LIN {X 0,Y 361.896,Z 471.407,A -85,B 0,C 180,E1 -13251.652,E2 -13251.652} C_VEL
LIN {X 0,Y 361.932,Z 471.4,A -85,B 0,C 180,E1 -13255.29,E2 -13255.29} C_VEL
LIN {X 0,Y 361.912,Z 471.406,A -85,B 0,C 180,E1 -13257.779,E2 -13257.779} C_VEL
LIN {X 0,Y 361.841,Z 471.415,A -85,B 0,C 180,E1 -13261.629,E2 -13261.629} C_VEL
LIN {X 0,Y 361.878,Z 471.407,A -85,B 0,C 180,E1 -13265.344,E2 -13265.344} C_VEL
LIN {X 0,Y 361.873,Z 471.407,A -85,B 0,C 180,E1 -13269.026,E2 -13269.026} C_VEL
LIN {X 0,Y 361.839,Z 471.41,A -85,B 0,C 180,E1 -13272.828,E2 -13272.828} C_VEL
LIN {X 0,Y 361.819,Z 471.417,A -85,B 0,C 180,E1 -13275.6,E2 -13275.6} C_VEL
LIN {X 0,Y 361.188,Z 471.501,A -85,B 0,C 180,E1 -13276.53,E2 -13276.53} C_VEL
LIN {X 0,Y 358.309,Z 471.855,A -85,B 0,C 180,E1 -13278.041,E2 -13278.041} C_VEL
LIN {X 0,Y 355.876,Z 472.155,A -85,B 0,C 180,E1 -13279.265,E2 -13279.265} C_VEL
LIN {X 0,Y 354.876,Z 472.279,A -85,B 0,C 180,E1 -13280.212,E2 -13280.212} C_VEL
LIN {X 0,Y 354.821,Z 472.284,A -85,B 0,C 180,E1 -13280.532,E2 -13280.532} C_VEL
LIN {X 0,Y 354.824,Z 472.285,A -85,B 0,C 180,E1 -13284.3,E2 -13284.3} C_VEL
LIN {X 0,Y 354.789,Z 472.294,A -85,B 0,C 180,E1 -13287.666,E2 -13287.666} C_VEL
LIN {X 0,Y 354.87,Z 472.278,A -85,B 0,C 180,E1 -13290.621,E2 -13290.621} C_VEL
LIN {X 0,Y 354.901,Z 472.276,A -85,B 0,C 180,E1 -13294.172,E2 -13294.172} C_VEL
LIN {X 0,Y 354.836,Z 472.286,A -85,B 0,C 180,E1 -13297.894,E2 -13297.894} C_VEL
LIN {X 0,Y 354.924,Z 472.275,A -85,B 0,C 180,E1 -13301.891,E2 -13301.891} C_VEL
LIN {X 0,Y 354.944,Z 472.272,A -85,B 0,C 180,E1 -13305.981,E2 -13305.981} C_VEL
LIN {X 0,Y 354.979,Z 472.269,A -85,B 0,C 180,E1 -13309.736,E2 -13309.736} C_VEL
LIN {X 0,Y 355.115,Z 472.25,A -85,B 0,C 180,E1 -13312.037,E2 -13312.037} C_VEL
LIN {X 0,Y 355.093,Z 472.251,A -85,B 0,C 180,E1 -13314.32,E2 -13314.32} C_VEL
LIN {X 0,Y 355.246,Z 472.236,A -85,B 0,C 180,E1 -13317.732,E2 -13317.732} C_VEL
LIN {X 0,Y 355.398,Z 472.214,A -85,B 0,C 180,E1 -13320,E2 -13320} C_VEL
LIN {X 0,Y 355.244,Z 472.232,A -85,B 0,C 180,E1 -13322.267,E2 -13322.267} C_VEL
LIN {X 0,Y 355.139,Z 472.246,A -85,B 0,C 180,E1 -13326.819,E2 -13326.819} C_VEL
LIN {X 0,Y 355.015,Z 472.263,A -85,B 0,C 180,E1 -13329.112,E2 -13329.112} C_VEL
LIN {X 0,Y 354.921,Z 472.272,A -85,B 0,C 180,E1 -13332.581,E2 -13332.581} C_VEL
LIN {X 0,Y 354.89,Z 472.276,A -85,B 0,C 180,E1 -13336.096,E2 -13336.096} C_VEL
LIN {X 0,Y 354.901,Z 472.274,A -85,B 0,C 180,E1 -13338.472,E2 -13338.472} C_VEL
LIN {X 0,Y 354.835,Z 472.283,A -85,B 0,C 180,E1 -13342.106,E2 -13342.106} C_VEL
LIN {X 0,Y 354.899,Z 472.276,A -85,B 0,C 180,E1 -13345.827,E2 -13345.827} C_VEL
LIN {X 0,Y 354.817,Z 472.288,A -85,B 0,C 180,E1 -13349.682,E2 -13349.682} C_VEL
LIN {X 0,Y 354.805,Z 472.289,A -85,B 0,C 180,E1 -13353.702,E2 -13353.702} C_VEL
LIN {X 0,Y 354.801,Z 472.287,A -85,B 0,C 180,E1 -13356.459,E2 -13356.459} C_VEL
LIN {X 0,Y 354.824,Z 472.288,A -85,B 0,C 180,E1 -13359.424,E2 -13359.424} C_VEL
LIN {X 0,Y 354.835,Z 472.285,A -85,B 0,C 180,E1 -13362.876,E2 -13362.876} C_VEL
LIN {X 0,Y 354.861,Z 472.442,A -85,B 0,C 180,E1 -13365.478,E2 -13365.478} C_VEL
LIN {X 0,Y 356.023,Z 478.787,A -85,B 0,C 180,E1 -13369.351,E2 -13369.351} C_VEL
LIN {X 0,Y 357.063,Z 485.29,A -85,B 0,C 180,E1 -13373.108,E2 -13373.108} C_VEL
LIN {X 0,Y 356.927,Z 489.111,A -85,B 0,C 180,E1 -13375.179,E2 -13375.179} C_VEL
LIN {X 0,Y 356.106,Z 495.602,A -85,B 0,C 180,E1 -13378.579,E2 -13378.579} C_VEL
LIN {X 0,Y 355.345,Z 502.874,A -85,B 0,C 180,E1 -13382.305,E2 -13382.305} C_VEL
LIN {X 0,Y 354.675,Z 509.674,A -85,B 0,C 180,E1 -13385.714,E2 -13385.714} C_VEL
LIN {X 0,Y 354.097,Z 517.685,A -85,B 0,C 180,E1 -13389.676,E2 -13389.676} C_VEL
LIN {X 0,Y 353.998,Z 519.753,A -85,B 0,C 180,E1 -13390.691,E2 -13390.691} C_VEL
LIN {X 0,Y 355.817,Z 535.091,A -85,B 0,C 180,E1 -13391.457,E2 -13391.457} C_VEL
LIN {X 0,Y 357.371,Z 548.346,A -85,B 0,C 180,E1 -13392.345,E2 -13392.345} C_VEL
LIN {X 0,Y 357.95,Z 556.63,A -85,B 0,C 180,E1 -13393.019,E2 -13393.019} C_VEL
LIN {X 0,Y 357.02,Z 568.5,A -85,B 0,C 180,E1 -13394.15,E2 -13394.15} C_VEL
LIN {X 0,Y 356.03,Z 579.361,A -85,B 0,C 180,E1 -13395.443,E2 -13395.443} C_VEL
LIN {X 0,Y 355.222,Z 588.935,A -85,B 0,C 180,E1 -13396.849,E2 -13396.849} C_VEL
LIN {X 0,Y 354.587,Z 596.98,A -85,B 0,C 180,E1 -13398.279,E2 -13398.279} C_VEL
LIN {X 0,Y 354.005,Z 604.908,A -85,B 0,C 180,E1 -13399.997,E2 -13399.997} C_VEL
LIN {X 0,Y 353.691,Z 610.279,A -85,B 0,C 180,E1 -13401.43,E2 -13401.43} C_VEL
LIN {X 0,Y 353.5,Z 615.518,A -85,B 0,C 180,E1 -13403.149,E2 -13403.149} C_VEL
LIN {X 0,Y 353.454,Z 619.542,A -85,B 0,C 180,E1 -13404.867,E2 -13404.867} C_VEL
LIN {X 0,Y 353.343,Z 622.453,A -85,B 0,C 180,E1 -13406.579,E2 -13406.579} C_VEL
LIN {X 0,Y 353.477,Z 623.816,A -85,B 0,C 180,E1 -13407.721,E2 -13407.721} C_VEL
LIN {X 0,Y 353.476,Z 624.737,A -85,B 0,C 180,E1 -13408.861,E2 -13408.861} C_VEL
LIN {X 0,Y 353.463,Z 625.243,A -85,B 0,C 180,E1 -13410,E2 -13410} C_VEL
LIN {X 0,Y 353.464,Z 625.318,A -85,B 0,C 180,E1 -13411.14,E2 -13411.14} C_VEL
LIN {X 0,Y 353.371,Z 624.931,A -85,B 0,C 180,E1 -13412.28,E2 -13412.28} C_VEL
LIN {X 0,Y 353.322,Z 622.937,A -85,B 0,C 180,E1 -13414.564,E2 -13414.564} C_VEL
LIN {X 0,Y 353.314,Z 620.847,A -85,B 0,C 180,E1 -13415.966,E2 -13415.966} C_VEL
LIN {X 0,Y 353.604,Z 616.652,A -85,B 0,C 180,E1 -13417.998,E2 -13417.998} C_VEL
LIN {X 0,Y 353.981,Z 611.938,A -85,B 0,C 180,E1 -13419.716,E2 -13419.716} C_VEL
LIN {X 0,Y 354.771,Z 604.943,A -85,B 0,C 180,E1 -13421.716,E2 -13421.716} C_VEL
LIN {X 0,Y 355.788,Z 597.461,A -85,B 0,C 180,E1 -13423.421,E2 -13423.421} C_VEL
LIN {X 0,Y 356.862,Z 588.946,A -85,B 0,C 180,E1 -13425.028,E2 -13425.028} C_VEL
LIN {X 0,Y 358.555,Z 578.253,A -85,B 0,C 180,E1 -13426.659,E2 -13426.659} C_VEL
LIN {X 0,Y 360.253,Z 567.141,A -85,B 0,C 180,E1 -13428.041,E2 -13428.041} C_VEL
LIN {X 0,Y 361.219,Z 559.295,A -85,B 0,C 180,E1 -13428.873,E2 -13428.873} C_VEL
LIN {X 0,Y 361.174,Z 546.774,A -85,B 0,C 180,E1 -13430.1,E2 -13430.1} C_VEL
LIN {X 0,Y 359.932,Z 535.75,A -85,B 0,C 180,E1 -13431.118,E2 -13431.118} C_VEL
LIN {X 0,Y 357.617,Z 524.701,A -85,B 0,C 180,E1 -13432.098,E2 -13432.098} C_VEL
LIN {X 0,Y 355.357,Z 517.035,A -85,B 0,C 180,E1 -13432.792,E2 -13432.792} C_VEL
LIN {X 0,Y 354.616,Z 513.908,A -85,B 0,C 180,E1 -13433.055,E2 -13433.055} C_VEL
LIN {X 0,Y 355.282,Z 507.666,A -85,B 0,C 180,E1 -13436.429,E2 -13436.429} C_VEL
LIN {X 0,Y 356.057,Z 502.051,A -85,B 0,C 180,E1 -13439.716,E2 -13439.716} C_VEL
LIN {X 0,Y 356.726,Z 498.243,A -85,B 0,C 180,E1 -13442.137,E2 -13442.137} C_VEL
LIN {X 0,Y 357.445,Z 494.507,A -85,B 0,C 180,E1 -13444.764,E2 -13444.764} C_VEL
LIN {X 0,Y 357.796,Z 492.467,A -85,B 0,C 180,E1 -13446.357,E2 -13446.357} C_VEL
LIN {X 0,Y 357.78,Z 489.641,A -85,B 0,C 180,E1 -13448.946,E2 -13448.946} C_VEL
LIN {X 0,Y 357.413,Z 487.044,A -85,B 0,C 180,E1 -13451.956,E2 -13451.956} C_VEL
LIN {X 0,Y 357.086,Z 485.013,A -85,B 0,C 180,E1 -13455.116,E2 -13455.116} C_VEL
LIN {X 0,Y 356.777,Z 483.627,A -85,B 0,C 180,E1 -13458.465,E2 -13458.465} C_VEL
LIN {X 0,Y 356.561,Z 482.938,A -85,B 0,C 180,E1 -13462.039,E2 -13462.039} C_VEL
LIN {X 0,Y 356.269,Z 482.954,A -85,B 0,C 180,E1 -13465.105,E2 -13465.105} C_VEL
LIN {X 0,Y 355.925,Z 483.444,A -85,B 0,C 180,E1 -13468.111,E2 -13468.111} C_VEL
LIN {X 0,Y 355.416,Z 484.534,A -85,B 0,C 180,E1 -13471.668,E2 -13471.668} C_VEL
LIN {X 0,Y 354.986,Z 486.226,A -85,B 0,C 180,E1 -13475.604,E2 -13475.604} C_VEL
LIN {X 0,Y 354.856,Z 487.017,A -85,B 0,C 180,E1 -13477.145,E2 -13477.145} C_VEL
LIN {X 0,Y 355.852,Z 489.82,A -85,B 0,C 180,E1 -13477.439,E2 -13477.439} C_VEL
LIN {X 0,Y 357.99,Z 494.025,A -85,B 0,C 180,E1 -13477.965,E2 -13477.965} C_VEL
LIN {X 0,Y 361.932,Z 504.222,A -85,B 0,C 180,E1 -13479.157,E2 -13479.157} C_VEL
LIN {X 0,Y 364.472,Z 513.793,A -85,B 0,C 180,E1 -13480.259,E2 -13480.259} C_VEL
LIN {X 0,Y 364.253,Z 518.028,A -85,B 0,C 180,E1 -13480.651,E2 -13480.651} C_VEL
LIN {X 0,Y 362.785,Z 529.035,A -85,B 0,C 180,E1 -13481.74,E2 -13481.74} C_VEL
LIN {X 0,Y 361.233,Z 539.619,A -85,B 0,C 180,E1 -13483.032,E2 -13483.032} C_VEL
LIN {X 0,Y 359.697,Z 548.878,A -85,B 0,C 180,E1 -13484.416,E2 -13484.416} C_VEL
LIN {X 0,Y 358.425,Z 556.592,A -85,B 0,C 180,E1 -13485.812,E2 -13485.812} C_VEL
LIN {X 0,Y 357.08,Z 564.286,A -85,B 0,C 180,E1 -13487.497,E2 -13487.497} C_VEL
LIN {X 0,Y 356.143,Z 570.486,A -85,B 0,C 180,E1 -13489.195,E2 -13489.195} C_VEL
LIN {X 0,Y 355.273,Z 575.452,A -85,B 0,C 180,E1 -13490.895,E2 -13490.895} C_VEL
LIN {X 0,Y 354.489,Z 579.713,A -85,B 0,C 180,E1 -13492.792,E2 -13492.792} C_VEL
LIN {X 0,Y 354.101,Z 582.167,A -85,B 0,C 180,E1 -13494.305,E2 -13494.305} C_VEL
LIN {X 0,Y 354.036,Z 583.522,A -85,B 0,C 180,E1 -13495.446,E2 -13495.446} C_VEL
LIN {X 0,Y 353.821,Z 584.446,A -85,B 0,C 180,E1 -13496.584,E2 -13496.584} C_VEL
LIN {X 0,Y 353.65,Z 584.978,A -85,B 0,C 180,E1 -13497.722,E2 -13497.722} C_VEL
LIN {X 0,Y 353.526,Z 585.118,A -85,B 0,C 180,E1 -13498.861,E2 -13498.861} C_VEL
LIN {X 0,Y 353.466,Z 584.834,A -85,B 0,C 180,E1 -13500,E2 -13500} C_VEL
LIN {X 0,Y 353.486,Z 584.117,A -85,B 0,C 180,E1 -13501.14,E2 -13501.14} C_VEL
LIN {X 0,Y 353.519,Z 583.003,A -85,B 0,C 180,E1 -13502.279,E2 -13502.279} C_VEL
LIN {X 0,Y 353.539,Z 580.526,A -85,B 0,C 180,E1 -13503.99,E2 -13503.99} C_VEL
LIN {X 0,Y 353.757,Z 577.033,A -85,B 0,C 180,E1 -13505.701,E2 -13505.701} C_VEL
LIN {X 0,Y 354.05,Z 572.439,A -85,B 0,C 180,E1 -13507.413,E2 -13507.413} C_VEL
LIN {X 0,Y 354.437,Z 566.619,A -85,B 0,C 180,E1 -13509.128,E2 -13509.128} C_VEL
LIN {X 0,Y 355.01,Z 559.372,A -85,B 0,C 180,E1 -13510.84,E2 -13510.84} C_VEL
LIN {X 0,Y 355.731,Z 550.381,A -85,B 0,C 180,E1 -13512.552,E2 -13512.552} C_VEL
LIN {X 0,Y 356.656,Z 540.246,A -85,B 0,C 180,E1 -13514.114,E2 -13514.114} C_VEL
LIN {X 0,Y 357.475,Z 529.945,A -85,B 0,C 180,E1 -13515.402,E2 -13515.402} C_VEL
LIN {X 0,Y 358.342,Z 517.407,A -85,B 0,C 180,E1 -13516.669,E2 -13516.669} C_VEL
LIN {X 0,Y 359.063,Z 507.592,A -85,B 0,C 180,E1 -13517.458,E2 -13517.458} C_VEL
LIN {X 0,Y 357.067,Z 496.682,A -85,B 0,C 180,E1 -13518.254,E2 -13518.254} C_VEL
LIN {X 0,Y 354.036,Z 482.545,A -85,B 0,C 180,E1 -13519.063,E2 -13519.063} C_VEL
LIN {X 0,Y 353.631,Z 480.363,A -85,B 0,C 180,E1 -13519.199,E2 -13519.199} C_VEL
LIN {X 0,Y 353.639,Z 477.42,A -85,B 0,C 180,E1 -13522.185,E2 -13522.185} C_VEL
LIN {X 0,Y 353.81,Z 473.84,A -85,B 0,C 180,E1 -13525.913,E2 -13525.913} C_VEL
LIN {X 0,Y 353.84,Z 472.639,A -85,B 0,C 180,E1 -13527.183,E2 -13527.183} C_VEL
LIN {X 0,Y 354.095,Z 472.378,A -85,B 0,C 180,E1 -13529.749,E2 -13529.749} C_VEL
LIN {X 0,Y 354.394,Z 472.343,A -85,B 0,C 180,E1 -13532.374,E2 -13532.374} C_VEL
LIN {X 0,Y 354.715,Z 472.299,A -85,B 0,C 180,E1 -13535.675,E2 -13535.675} C_VEL
LIN {X 0,Y 354.797,Z 472.29,A -85,B 0,C 180,E1 -13537.885,E2 -13537.885} C_VEL
LIN {X 0,Y 354.792,Z 472.288,A -85,B 0,C 180,E1 -13541.172,E2 -13541.172} C_VEL
LIN {X 0,Y 354.768,Z 472.294,A -85,B 0,C 180,E1 -13544.507,E2 -13544.507} C_VEL
LIN {X 0,Y 354.799,Z 472.288,A -85,B 0,C 180,E1 -13547.663,E2 -13547.663} C_VEL
LIN {X 0,Y 354.819,Z 472.287,A -85,B 0,C 180,E1 -13550.666,E2 -13550.666} C_VEL
LIN {X 0,Y 354.827,Z 472.288,A -85,B 0,C 180,E1 -13554.301,E2 -13554.301} C_VEL
LIN {X 0,Y 354.792,Z 472.29,A -85,B 0,C 180,E1 -13557.667,E2 -13557.667} C_VEL
LIN {X 0,Y 354.851,Z 472.282,A -85,B 0,C 180,E1 -13561.619,E2 -13561.619} C_VEL
LIN {X 0,Y 354.904,Z 472.279,A -85,B 0,C 180,E1 -13564.173,E2 -13564.173} C_VEL
LIN {X 0,Y 354.84,Z 472.285,A -85,B 0,C 180,E1 -13567.894,E2 -13567.894} C_VEL
LIN {X 0,Y 354.928,Z 472.275,A -85,B 0,C 180,E1 -13571.891,E2 -13571.891} C_VEL
LIN {X 0,Y 354.948,Z 472.274,A -85,B 0,C 180,E1 -13575.981,E2 -13575.981} C_VEL
LIN {X 0,Y 354.982,Z 472.268,A -85,B 0,C 180,E1 -13579.736,E2 -13579.736} C_VEL
LIN {X 0,Y 355.125,Z 472.246,A -85,B 0,C 180,E1 -13583.18,E2 -13583.18} C_VEL
LIN {X 0,Y 355.249,Z 472.235,A -85,B 0,C 180,E1 -13587.732,E2 -13587.732} C_VEL
LIN {X 0,Y 355.401,Z 472.217,A -85,B 0,C 180,E1 -13590,E2 -13590} C_VEL
LIN {X 0,Y 355.249,Z 472.235,A -85,B 0,C 180,E1 -13592.267,E2 -13592.267} C_VEL
LIN {X 0,Y 355.108,Z 472.248,A -85,B 0,C 180,E1 -13596.82,E2 -13596.82} C_VEL
LIN {X 0,Y 354.983,Z 472.267,A -85,B 0,C 180,E1 -13600.264,E2 -13600.264} C_VEL
LIN {X 0,Y 354.947,Z 472.273,A -85,B 0,C 180,E1 -13604.019,E2 -13604.019} C_VEL
LIN {X 0,Y 354.927,Z 472.275,A -85,B 0,C 180,E1 -13608.108,E2 -13608.108} C_VEL
LIN {X 0,Y 354.839,Z 472.286,A -85,B 0,C 180,E1 -13612.106,E2 -13612.106} C_VEL
LIN {X 0,Y 354.903,Z 472.279,A -85,B 0,C 180,E1 -13615.827,E2 -13615.827} C_VEL
LIN {X 0,Y 354.821,Z 472.289,A -85,B 0,C 180,E1 -13619.681,E2 -13619.681} C_VEL
LIN {X 0,Y 354.809,Z 472.29,A -85,B 0,C 180,E1 -13623.702,E2 -13623.702} C_VEL
LIN {X 0,Y 354.804,Z 472.287,A -85,B 0,C 180,E1 -13626.458,E2 -13626.458} C_VEL
LIN {X 0,Y 354.826,Z 472.287,A -85,B 0,C 180,E1 -13629.423,E2 -13629.423} C_VEL
LIN {X 0,Y 354.791,Z 472.288,A -85,B 0,C 180,E1 -13632.867,E2 -13632.867} C_VEL
LIN {X 0,Y 354.771,Z 472.294,A -85,B 0,C 180,E1 -13636.103,E2 -13636.103} C_VEL
LIN {X 0,Y 354.79,Z 472.289,A -85,B 0,C 180,E1 -13639.179,E2 -13639.179} C_VEL
LIN {X 0,Y 354.821,Z 472.284,A -85,B 0,C 180,E1 -13640.532,E2 -13640.532} C_VEL
LIN {X 0,Y 354.218,Z 472.366,A -85,B 0,C 180,E1 -13641.48,E2 -13641.48} C_VEL
LIN {X 0,Y 351.361,Z 472.727,A -85,B 0,C 180,E1 -13643.02,E2 -13643.02} C_VEL
LIN {X 0,Y 348.896,Z 473.032,A -85,B 0,C 180,E1 -13644.267,E2 -13644.267} C_VEL
LIN {X 0,Y 347.832,Z 473.161,A -85,B 0,C 180,E1 -13645.232,E2 -13645.232} C_VEL
LIN {X 0,Y 347.746,Z 473.17,A -85,B 0,C 180,E1 -13645.559,E2 -13645.559} C_VEL
LIN {X 0,Y 347.765,Z 473.168,A -85,B 0,C 180,E1 -13649.653,E2 -13649.653} C_VEL
LIN {X 0,Y 347.853,Z 473.152,A -85,B 0,C 180,E1 -13652.744,E2 -13652.744} C_VEL
LIN {X 0,Y 347.79,Z 473.162,A -85,B 0,C 180,E1 -13656.162,E2 -13656.162} C_VEL
LIN {X 0,Y 347.819,Z 473.159,A -85,B 0,C 180,E1 -13659.909,E2 -13659.909} C_VEL
LIN {X 0,Y 347.868,Z 473.151,A -85,B 0,C 180,E1 -13662.359,E2 -13662.359} C_VEL
LIN {X 0,Y 347.898,Z 473.149,A -85,B 0,C 180,E1 -13665.97,E2 -13665.97} C_VEL
LIN {X 0,Y 347.929,Z 473.148,A -85,B 0,C 180,E1 -13669.525,E2 -13669.525} C_VEL
LIN {X 0,Y 348.075,Z 473.128,A -85,B 0,C 180,E1 -13671.874,E2 -13671.874} C_VEL
LIN {X 0,Y 348.068,Z 473.126,A -85,B 0,C 180,E1 -13674.205,E2 -13674.205} C_VEL
LIN {X 0,Y 348.209,Z 473.112,A -85,B 0,C 180,E1 -13677.686,E2 -13677.686} C_VEL
LIN {X 0,Y 348.347,Z 473.092,A -85,B 0,C 180,E1 -13680,E2 -13680} C_VEL
LIN {X 0,Y 348.207,Z 473.108,A -85,B 0,C 180,E1 -13682.313,E2 -13682.313} C_VEL
LIN {X 0,Y 348.107,Z 473.122,A -85,B 0,C 180,E1 -13686.957,E2 -13686.957} C_VEL
LIN {X 0,Y 347.968,Z 473.142,A -85,B 0,C 180,E1 -13689.298,E2 -13689.298} C_VEL
LIN {X 0,Y 347.89,Z 473.149,A -85,B 0,C 180,E1 -13692.839,E2 -13692.839} C_VEL
LIN {X 0,Y 347.839,Z 473.154,A -85,B 0,C 180,E1 -13696.431,E2 -13696.431} C_VEL
LIN {X 0,Y 347.851,Z 473.154,A -85,B 0,C 180,E1 -13698.86,E2 -13698.86} C_VEL
LIN {X 0,Y 347.774,Z 473.162,A -85,B 0,C 180,E1 -13702.579,E2 -13702.579} C_VEL
LIN {X 0,Y 347.813,Z 473.16,A -85,B 0,C 180,E1 -13705.108,E2 -13705.108} C_VEL
LIN {X 0,Y 347.808,Z 473.161,A -85,B 0,C 180,E1 -13707.694,E2 -13707.694} C_VEL
LIN {X 0,Y 347.749,Z 473.165,A -85,B 0,C 180,E1 -13710.348,E2 -13710.348} C_VEL
LIN {X 0,Y 347.748,Z 473.166,A -85,B 0,C 180,E1 -13714.044,E2 -13714.044} C_VEL
LIN {X 0,Y 347.766,Z 473.168,A -85,B 0,C 180,E1 -13717.32,E2 -13717.32} C_VEL
LIN {X 0,Y 347.793,Z 473.16,A -85,B 0,C 180,E1 -13720.289,E2 -13720.289} C_VEL
LIN {X 0,Y 347.786,Z 473.166,A -85,B 0,C 180,E1 -13723.398,E2 -13723.398} C_VEL
LIN {X 0,Y 347.86,Z 473.23,A -85,B 0,C 180,E1 -13725.206,E2 -13725.206} C_VEL
LIN {X 0,Y 348.936,Z 479.491,A -85,B 0,C 180,E1 -13729.112,E2 -13729.112} C_VEL
LIN {X 0,Y 349.857,Z 484.863,A -85,B 0,C 180,E1 -13732.299,E2 -13732.299} C_VEL
LIN {X 0,Y 349.979,Z 488.554,A -85,B 0,C 180,E1 -13734.384,E2 -13734.384} C_VEL
LIN {X 0,Y 349.225,Z 494.695,A -85,B 0,C 180,E1 -13737.697,E2 -13737.697} C_VEL
LIN {X 0,Y 348.389,Z 502.297,A -85,B 0,C 180,E1 -13741.702,E2 -13741.702} C_VEL
LIN {X 0,Y 347.642,Z 509.619,A -85,B 0,C 180,E1 -13745.468,E2 -13745.468} C_VEL
LIN {X 0,Y 346.993,Z 518.291,A -85,B 0,C 180,E1 -13749.86,E2 -13749.86} C_VEL
LIN {X 0,Y 346.912,Z 519.429,A -85,B 0,C 180,E1 -13750.434,E2 -13750.434} C_VEL
LIN {X 0,Y 348.644,Z 534.247,A -85,B 0,C 180,E1 -13751.184,E2 -13751.184} C_VEL
LIN {X 0,Y 350.184,Z 547.739,A -85,B 0,C 180,E1 -13752.107,E2 -13752.107} C_VEL
LIN {X 0,Y 350.889,Z 557.922,A -85,B 0,C 180,E1 -13752.967,E2 -13752.967} C_VEL
LIN {X 0,Y 349.929,Z 569.441,A -85,B 0,C 180,E1 -13754.119,E2 -13754.119} C_VEL
LIN {X 0,Y 348.815,Z 580.976,A -85,B 0,C 180,E1 -13755.572,E2 -13755.572} C_VEL
LIN {X 0,Y 348.09,Z 589.406,A -85,B 0,C 180,E1 -13756.872,E2 -13756.872} C_VEL
LIN {X 0,Y 347.451,Z 597.304,A -85,B 0,C 180,E1 -13758.33,E2 -13758.33} C_VEL
LIN {X 0,Y 346.91,Z 605.057,A -85,B 0,C 180,E1 -13760.084,E2 -13760.084} C_VEL
LIN {X 0,Y 346.541,Z 611.261,A -85,B 0,C 180,E1 -13761.839,E2 -13761.839} C_VEL
LIN {X 0,Y 346.342,Z 616.887,A -85,B 0,C 180,E1 -13763.887,E2 -13763.887} C_VEL
LIN {X 0,Y 346.366,Z 619.905,A -85,B 0,C 180,E1 -13765.345,E2 -13765.345} C_VEL
LIN {X 0,Y 346.266,Z 621.792,A -85,B 0,C 180,E1 -13766.509,E2 -13766.509} C_VEL
LIN {X 0,Y 346.397,Z 623.234,A -85,B 0,C 180,E1 -13767.675,E2 -13767.675} C_VEL
LIN {X 0,Y 346.414,Z 624.197,A -85,B 0,C 180,E1 -13768.838,E2 -13768.838} C_VEL
LIN {X 0,Y 346.399,Z 624.74,A -85,B 0,C 180,E1 -13770,E2 -13770} C_VEL
LIN {X 0,Y 346.4,Z 624.872,A -85,B 0,C 180,E1 -13771.163,E2 -13771.163} C_VEL
LIN {X 0,Y 346.272,Z 624.543,A -85,B 0,C 180,E1 -13772.327,E2 -13772.327} C_VEL
LIN {X 0,Y 346.215,Z 623.786,A -85,B 0,C 180,E1 -13773.492,E2 -13773.492} C_VEL
LIN {X 0,Y 346.233,Z 622.625,A -85,B 0,C 180,E1 -13774.657,E2 -13774.657} C_VEL
LIN {X 0,Y 346.242,Z 620.845,A -85,B 0,C 180,E1 -13775.957,E2 -13775.957} C_VEL
LIN {X 0,Y 346.544,Z 616.518,A -85,B 0,C 180,E1 -13778.162,E2 -13778.162} C_VEL
LIN {X 0,Y 346.965,Z 611.913,A -85,B 0,C 180,E1 -13779.914,E2 -13779.914} C_VEL
LIN {X 0,Y 347.817,Z 605.087,A -85,B 0,C 180,E1 -13781.953,E2 -13781.953} C_VEL
LIN {X 0,Y 348.887,Z 597.774,A -85,B 0,C 180,E1 -13783.692,E2 -13783.692} C_VEL
LIN {X 0,Y 350.175,Z 588.755,A -85,B 0,C 180,E1 -13785.451,E2 -13785.451} C_VEL
LIN {X 0,Y 351.97,Z 578.118,A -85,B 0,C 180,E1 -13787.129,E2 -13787.129} C_VEL
LIN {X 0,Y 353.797,Z 567.069,A -85,B 0,C 180,E1 -13788.532,E2 -13788.532} C_VEL
LIN {X 0,Y 354.704,Z 559.366,A -85,B 0,C 180,E1 -13789.383,E2 -13789.383} C_VEL
LIN {X 0,Y 354.764,Z 547.801,A -85,B 0,C 180,E1 -13790.583,E2 -13790.583} C_VEL
LIN {X 0,Y 353.472,Z 536.234,A -85,B 0,C 180,E1 -13791.711,E2 -13791.711} C_VEL
LIN {X 0,Y 350.89,Z 524.202,A -85,B 0,C 180,E1 -13792.878,E2 -13792.878} C_VEL
LIN {X 0,Y 348.41,Z 516.176,A -85,B 0,C 180,E1 -13793.663,E2 -13793.663} C_VEL
LIN {X 0,Y 347.741,Z 513.187,A -85,B 0,C 180,E1 -13793.94,E2 -13793.94} C_VEL
LIN {X 0,Y 348.508,Z 506.68,A -85,B 0,C 180,E1 -13797.634,E2 -13797.634} C_VEL
LIN {X 0,Y 349.533,Z 500.482,A -85,B 0,C 180,E1 -13801.519,E2 -13801.519} C_VEL
LIN {X 0,Y 350.446,Z 496.008,A -85,B 0,C 180,E1 -13804.691,E2 -13804.691} C_VEL
LIN {X 0,Y 350.87,Z 493.249,A -85,B 0,C 180,E1 -13806.935,E2 -13806.935} C_VEL
LIN {X 0,Y 350.879,Z 491.449,A -85,B 0,C 180,E1 -13808.633,E2 -13808.633} C_VEL
LIN {X 0,Y 350.474,Z 488.488,A -85,B 0,C 180,E1 -13812.102,E2 -13812.102} C_VEL
LIN {X 0,Y 350.142,Z 486.451,A -85,B 0,C 180,E1 -13815.371,E2 -13815.371} C_VEL
LIN {X 0,Y 349.864,Z 485.181,A -85,B 0,C 180,E1 -13818.479,E2 -13818.479} C_VEL
LIN {X 0,Y 349.634,Z 484.512,A -85,B 0,C 180,E1 -13821.623,E2 -13821.623} C_VEL
LIN {X 0,Y 349.398,Z 484.393,A -85,B 0,C 180,E1 -13824.315,E2 -13824.315} C_VEL
LIN {X 0,Y 349.006,Z 484.796,A -85,B 0,C 180,E1 -13827.754,E2 -13827.754} C_VEL
LIN {X 0,Y 348.523,Z 485.683,A -85,B 0,C 180,E1 -13831.056,E2 -13831.056} C_VEL
LIN {X 0,Y 348.058,Z 487.19,A -85,B 0,C 180,E1 -13834.911,E2 -13834.911} C_VEL
LIN {X 0,Y 347.955,Z 487.974,A -85,B 0,C 180,E1 -13836.278,E2 -13836.278} C_VEL
LIN {X 0,Y 349.083,Z 490.882,A -85,B 0,C 180,E1 -13836.62,E2 -13836.62} C_VEL
LIN {X 0,Y 350.066,Z 492.672,A -85,B 0,C 180,E1 -13836.876,E2 -13836.876} C_VEL
LIN {X 0,Y 354.719,Z 503.244,A -85,B 0,C 180,E1 -13838.251,E2 -13838.251} C_VEL
LIN {X 0,Y 357.709,Z 513.477,A -85,B 0,C 180,E1 -13839.507,E2 -13839.507} C_VEL
LIN {X 0,Y 358.384,Z 516.83,A -85,B 0,C 180,E1 -13839.915,E2 -13839.915} C_VEL
LIN {X 0,Y 356.794,Z 528.176,A -85,B 0,C 180,E1 -13841.033,E2 -13841.033} C_VEL
LIN {X 0,Y 355.113,Z 538.661,A -85,B 0,C 180,E1 -13842.316,E2 -13842.316} C_VEL
LIN {X 0,Y 353.335,Z 548.893,A -85,B 0,C 180,E1 -13843.831,E2 -13843.831} C_VEL
LIN {X 0,Y 351.892,Z 556.682,A -85,B 0,C 180,E1 -13845.248,E2 -13845.248} C_VEL
LIN {X 0,Y 350.485,Z 564.358,A -85,B 0,C 180,E1 -13846.963,E2 -13846.963} C_VEL
LIN {X 0,Y 349.262,Z 571.565,A -85,B 0,C 180,E1 -13848.98,E2 -13848.98} C_VEL
LIN {X 0,Y 348.333,Z 576.413,A -85,B 0,C 180,E1 -13850.712,E2 -13850.712} C_VEL
LIN {X 0,Y 347.781,Z 579.211,A -85,B 0,C 180,E1 -13851.974,E2 -13851.974} C_VEL
LIN {X 0,Y 347.326,Z 581.16,A -85,B 0,C 180,E1 -13853.027,E2 -13853.027} C_VEL
LIN {X 0,Y 347.064,Z 582.881,A -85,B 0,C 180,E1 -13854.189,E2 -13854.189} C_VEL
LIN {X 0,Y 347.001,Z 584.138,A -85,B 0,C 180,E1 -13855.353,E2 -13855.353} C_VEL
LIN {X 0,Y 346.779,Z 585.014,A -85,B 0,C 180,E1 -13856.515,E2 -13856.515} C_VEL
LIN {X 0,Y 346.595,Z 585.498,A -85,B 0,C 180,E1 -13857.676,E2 -13857.676} C_VEL
LIN {X 0,Y 346.464,Z 585.579,A -85,B 0,C 180,E1 -13858.838,E2 -13858.838} C_VEL
LIN {X 0,Y 346.402,Z 585.211,A -85,B 0,C 180,E1 -13860,E2 -13860} C_VEL
LIN {X 0,Y 346.406,Z 584.444,A -85,B 0,C 180,E1 -13861.163,E2 -13861.163} C_VEL
LIN {X 0,Y 346.425,Z 583.279,A -85,B 0,C 180,E1 -13862.326,E2 -13862.326} C_VEL
LIN {X 0,Y 346.465,Z 580.708,A -85,B 0,C 180,E1 -13864.072,E2 -13864.072} C_VEL
LIN {X 0,Y 346.692,Z 577.123,A -85,B 0,C 180,E1 -13865.818,E2 -13865.818} C_VEL
LIN {X 0,Y 346.982,Z 572.433,A -85,B 0,C 180,E1 -13867.566,E2 -13867.566} C_VEL
LIN {X 0,Y 347.477,Z 565.339,A -85,B 0,C 180,E1 -13869.606,E2 -13869.606} C_VEL
LIN {X 0,Y 348.116,Z 557.685,A -85,B 0,C 180,E1 -13871.353,E2 -13871.353} C_VEL
LIN {X 0,Y 348.77,Z 549.935,A -85,B 0,C 180,E1 -13872.807,E2 -13872.807} C_VEL
LIN {X 0,Y 349.681,Z 539.547,A -85,B 0,C 180,E1 -13874.402,E2 -13874.402} C_VEL
LIN {X 0,Y 350.546,Z 529.042,A -85,B 0,C 180,E1 -13875.714,E2 -13875.714} C_VEL
LIN {X 0,Y 351.363,Z 517.771,A -85,B 0,C 180,E1 -13876.86,E2 -13876.86} C_VEL
LIN {X 0,Y 352.076,Z 508.198,A -85,B 0,C 180,E1 -13877.648,E2 -13877.648} C_VEL
LIN {X 0,Y 349.529,Z 495.098,A -85,B 0,C 180,E1 -13878.614,E2 -13878.614} C_VEL
LIN {X 0,Y 346.686,Z 481.525,A -85,B 0,C 180,E1 -13879.388,E2 -13879.388} C_VEL
LIN {X 0,Y 346.572,Z 480.711,A -85,B 0,C 180,E1 -13879.471,E2 -13879.471} C_VEL
LIN {X 0,Y 346.604,Z 477.601,A -85,B 0,C 180,E1 -13882.66,E2 -13882.66} C_VEL
LIN {X 0,Y 346.776,Z 473.976,A -85,B 0,C 180,E1 -13886.479,E2 -13886.479} C_VEL
LIN {X 0,Y 346.822,Z 473.287,A -85,B 0,C 180,E1 -13887.78,E2 -13887.78} C_VEL
LIN {X 0,Y 347.129,Z 473.248,A -85,B 0,C 180,E1 -13890.408,E2 -13890.408} C_VEL
LIN {X 0,Y 347.556,Z 473.194,A -85,B 0,C 180,E1 -13894.486,E2 -13894.486} C_VEL
LIN {X 0,Y 347.767,Z 473.166,A -85,B 0,C 180,E1 -13897.987,E2 -13897.987} C_VEL
LIN {X 0,Y 347.755,Z 473.167,A -85,B 0,C 180,E1 -13901.83,E2 -13901.83} C_VEL
LIN {X 0,Y 347.71,Z 473.17,A -85,B 0,C 180,E1 -13905.027,E2 -13905.027} C_VEL
LIN {X 0,Y 347.755,Z 473.169,A -85,B 0,C 180,E1 -13908.397,E2 -13908.397} C_VEL
LIN {X 0,Y 347.779,Z 473.166,A -85,B 0,C 180,E1 -13912.011,E2 -13912.011} C_VEL
LIN {X 0,Y 347.749,Z 473.166,A -85,B 0,C 180,E1 -13915.536,E2 -13915.536} C_VEL
LIN {X 0,Y 347.75,Z 473.17,A -85,B 0,C 180,E1 -13918.301,E2 -13918.301} C_VEL
LIN {X 0,Y 347.783,Z 473.161,A -85,B 0,C 180,E1 -13920.988,E2 -13920.988} C_VEL
LIN {X 0,Y 347.836,Z 473.156,A -85,B 0,C 180,E1 -13923.608,E2 -13923.608} C_VEL
LIN {X 0,Y 347.794,Z 473.165,A -85,B 0,C 180,E1 -13926.162,E2 -13926.162} C_VEL
LIN {X 0,Y 347.823,Z 473.16,A -85,B 0,C 180,E1 -13929.91,E2 -13929.91} C_VEL
LIN {X 0,Y 347.872,Z 473.153,A -85,B 0,C 180,E1 -13932.359,E2 -13932.359} C_VEL
LIN {X 0,Y 347.902,Z 473.151,A -85,B 0,C 180,E1 -13935.971,E2 -13935.971} C_VEL
LIN {X 0,Y 347.933,Z 473.144,A -85,B 0,C 180,E1 -13939.525,E2 -13939.525} C_VEL
LIN {X 0,Y 348.092,Z 473.122,A -85,B 0,C 180,E1 -13943.042,E2 -13943.042} C_VEL
LIN {X 0,Y 348.211,Z 473.111,A -85,B 0,C 180,E1 -13947.686,E2 -13947.686} C_VEL
LIN {X 0,Y 348.35,Z 473.096,A -85,B 0,C 180,E1 -13950,E2 -13950} C_VEL
LIN {X 0,Y 348.211,Z 473.111,A -85,B 0,C 180,E1 -13952.313,E2 -13952.313} C_VEL
LIN {X 0,Y 348.075,Z 473.124,A -85,B 0,C 180,E1 -13956.958,E2 -13956.958} C_VEL
LIN {X 0,Y 347.934,Z 473.144,A -85,B 0,C 180,E1 -13960.474,E2 -13960.474} C_VEL
LIN {X 0,Y 347.903,Z 473.15,A -85,B 0,C 180,E1 -13964.149,E2 -13964.149} C_VEL
LIN {X 0,Y 347.896,Z 473.149,A -85,B 0,C 180,E1 -13968.29,E2 -13968.29} C_VEL
LIN {X 0,Y 347.793,Z 473.163,A -85,B 0,C 180,E1 -13971.635,E2 -13971.635} C_VEL
LIN {X 0,Y 347.816,Z 473.157,A -85,B 0,C 180,E1 -13975.108,E2 -13975.108} C_VEL
LIN {X 0,Y 347.812,Z 473.162,A -85,B 0,C 180,E1 -13977.694,E2 -13977.694} C_VEL
LIN {X 0,Y 347.752,Z 473.166,A -85,B 0,C 180,E1 -13980.347,E2 -13980.347} C_VEL
LIN {X 0,Y 347.751,Z 473.168,A -85,B 0,C 180,E1 -13984.043,E2 -13984.043} C_VEL
LIN {X 0,Y 347.769,Z 473.164,A -85,B 0,C 180,E1 -13987.32,E2 -13987.32} C_VEL
LIN {X 0,Y 347.735,Z 473.168,A -85,B 0,C 180,E1 -13990.296,E2 -13990.296} C_VEL
LIN {X 0,Y 347.726,Z 473.17,A -85,B 0,C 180,E1 -13993.407,E2 -13993.407} C_VEL
LIN {X 0,Y 347.727,Z 473.168,A -85,B 0,C 180,E1 -13996.686,E2 -13996.686} C_VEL
LIN {X 0,Y 347.749,Z 473.167,A -85,B 0,C 180,E1 -14000.172,E2 -14000.172} C_VEL
LIN {X 0,Y 347.764,Z 473.163,A -85,B 0,C 180,E1 -14002.679,E2 -14002.679} C_VEL
LIN {X 0,Y 347.746,Z 473.17,A -85,B 0,C 180,E1 -14005.559,E2 -14005.559} C_VEL
LIN {X 0,Y 347.091,Z 473.248,A -85,B 0,C 180,E1 -14006.526,E2 -14006.526} C_VEL
LIN {X 0,Y 344.287,Z 473.598,A -85,B 0,C 180,E1 -14008.1,E2 -14008.1} C_VEL
LIN {X 0,Y 341.894,Z 473.897,A -85,B 0,C 180,E1 -14009.374,E2 -14009.374} C_VEL
LIN {X 0,Y 340.846,Z 474.026,A -85,B 0,C 180,E1 -14010.358,E2 -14010.358} C_VEL
LIN {X 0,Y 340.748,Z 474.037,A -85,B 0,C 180,E1 -14010.692,E2 -14010.692} C_VEL
LIN {X 0,Y 340.806,Z 474.031,A -85,B 0,C 180,E1 -14013.02,E2 -14013.02} C_VEL
LIN {X 0,Y 340.73,Z 474.04,A -85,B 0,C 180,E1 -14016.927,E2 -14016.927} C_VEL
LIN {X 0,Y 340.796,Z 474.031,A -85,B 0,C 180,E1 -14020.733,E2 -14020.733} C_VEL
LIN {X 0,Y 340.788,Z 474.035,A -85,B 0,C 180,E1 -14023.218,E2 -14023.218} C_VEL
LIN {X 0,Y 340.845,Z 474.026,A -85,B 0,C 180,E1 -14026.89,E2 -14026.89} C_VEL
LIN {X 0,Y 340.929,Z 474.015,A -85,B 0,C 180,E1 -14030.507,E2 -14030.507} C_VEL
LIN {X 0,Y 341.076,Z 473.997,A -85,B 0,C 180,E1 -14032.898,E2 -14032.898} C_VEL
LIN {X 0,Y 341.17,Z 473.989,A -85,B 0,C 180,E1 -14037.638,E2 -14037.638} C_VEL
LIN {X 0,Y 341.297,Z 473.97,A -85,B 0,C 180,E1 -14040,E2 -14040} C_VEL
LIN {X 0,Y 341.169,Z 473.985,A -85,B 0,C 180,E1 -14042.361,E2 -14042.361} C_VEL
LIN {X 0,Y 341.076,Z 473.999,A -85,B 0,C 180,E1 -14047.102,E2 -14047.102} C_VEL
LIN {X 0,Y 340.871,Z 474.022,A -85,B 0,C 180,E1 -14050.694,E2 -14050.694} C_VEL
LIN {X 0,Y 340.863,Z 474.023,A -85,B 0,C 180,E1 -14054.325,E2 -14054.325} C_VEL
LIN {X 0,Y 340.837,Z 474.026,A -85,B 0,C 180,E1 -14058.466,E2 -14058.466} C_VEL
LIN {X 0,Y 340.753,Z 474.038,A -85,B 0,C 180,E1 -14061.857,E2 -14061.857} C_VEL
LIN {X 0,Y 340.772,Z 474.037,A -85,B 0,C 180,E1 -14065.664,E2 -14065.664} C_VEL
LIN {X 0,Y 340.728,Z 474.04,A -85,B 0,C 180,E1 -14068.321,E2 -14068.321} C_VEL
LIN {X 0,Y 340.697,Z 474.047,A -85,B 0,C 180,E1 -14071.045,E2 -14071.045} C_VEL
LIN {X 0,Y 340.718,Z 474.046,A -85,B 0,C 180,E1 -14075.279,E2 -14075.279} C_VEL
LIN {X 0,Y 340.714,Z 474.041,A -85,B 0,C 180,E1 -14078.387,E2 -14078.387} C_VEL
LIN {X 0,Y 340.725,Z 474.045,A -85,B 0,C 180,E1 -14081.304,E2 -14081.304} C_VEL
LIN {X 0,Y 340.807,Z 474.138,A -85,B 0,C 180,E1 -14085.015,E2 -14085.015} C_VEL
LIN {X 0,Y 341.845,Z 480.171,A -85,B 0,C 180,E1 -14088.861,E2 -14088.861} C_VEL
LIN {X 0,Y 342.739,Z 485.393,A -85,B 0,C 180,E1 -14092.037,E2 -14092.037} C_VEL
LIN {X 0,Y 342.977,Z 487.975,A -85,B 0,C 180,E1 -14093.541,E2 -14093.541} C_VEL
LIN {X 0,Y 342.495,Z 493.006,A -85,B 0,C 180,E1 -14096.356,E2 -14096.356} C_VEL
LIN {X 0,Y 341.578,Z 500.48,A -85,B 0,C 180,E1 -14100.409,E2 -14100.409} C_VEL
LIN {X 0,Y 340.874,Z 506.647,A -85,B 0,C 180,E1 -14103.687,E2 -14103.687} C_VEL
LIN {X 0,Y 340.185,Z 513.997,A -85,B 0,C 180,E1 -14107.53,E2 -14107.53} C_VEL
LIN {X 0,Y 339.852,Z 519.087,A -85,B 0,C 180,E1 -14110.168,E2 -14110.168} C_VEL
LIN {X 0,Y 341.647,Z 534.983,A -85,B 0,C 180,E1 -14111.013,E2 -14111.013} C_VEL
LIN {X 0,Y 343.235,Z 548.914,A -85,B 0,C 180,E1 -14112.009,E2 -14112.009} C_VEL
LIN {X 0,Y 343.871,Z 557.458,A -85,B 0,C 180,E1 -14112.762,E2 -14112.762} C_VEL
LIN {X 0,Y 342.932,Z 568.97,A -85,B 0,C 180,E1 -14113.939,E2 -14113.939} C_VEL
LIN {X 0,Y 341.813,Z 580.04,A -85,B 0,C 180,E1 -14115.357,E2 -14115.357} C_VEL
LIN {X 0,Y 340.966,Z 589.793,A -85,B 0,C 180,E1 -14116.895,E2 -14116.895} C_VEL
LIN {X 0,Y 340.347,Z 597.551,A -85,B 0,C 180,E1 -14118.385,E2 -14118.385} C_VEL
LIN {X 0,Y 339.789,Z 605.148,A -85,B 0,C 180,E1 -14120.175,E2 -14120.175} C_VEL
LIN {X 0,Y 339.415,Z 612.167,A -85,B 0,C 180,E1 -14122.265,E2 -14122.265} C_VEL
LIN {X 0,Y 339.258,Z 616.773,A -85,B 0,C 180,E1 -14124.055,E2 -14124.055} C_VEL
LIN {X 0,Y 339.302,Z 619.183,A -85,B 0,C 180,E1 -14125.248,E2 -14125.248} C_VEL
LIN {X 0,Y 339.19,Z 621.11,A -85,B 0,C 180,E1 -14126.436,E2 -14126.436} C_VEL
LIN {X 0,Y 339.304,Z 622.62,A -85,B 0,C 180,E1 -14127.626,E2 -14127.626} C_VEL
LIN {X 0,Y 339.353,Z 623.646,A -85,B 0,C 180,E1 -14128.814,E2 -14128.814} C_VEL
LIN {X 0,Y 339.338,Z 624.231,A -85,B 0,C 180,E1 -14130,E2 -14130} C_VEL
LIN {X 0,Y 339.335,Z 624.403,A -85,B 0,C 180,E1 -14131.187,E2 -14131.187} C_VEL
LIN {X 0,Y 339.175,Z 624.149,A -85,B 0,C 180,E1 -14132.375,E2 -14132.375} C_VEL
LIN {X 0,Y 339.136,Z 623.445,A -85,B 0,C 180,E1 -14133.565,E2 -14133.565} C_VEL
LIN {X 0,Y 339.129,Z 622.325,A -85,B 0,C 180,E1 -14134.755,E2 -14134.755} C_VEL
LIN {X 0,Y 339.141,Z 620.8,A -85,B 0,C 180,E1 -14135.948,E2 -14135.948} C_VEL
LIN {X 0,Y 339.38,Z 617.682,A -85,B 0,C 180,E1 -14137.736,E2 -14137.736} C_VEL
LIN {X 0,Y 339.772,Z 613.538,A -85,B 0,C 180,E1 -14139.525,E2 -14139.525} C_VEL
LIN {X 0,Y 340.496,Z 607.337,A -85,B 0,C 180,E1 -14141.61,E2 -14141.61} C_VEL
LIN {X 0,Y 341.817,Z 599.411,A -85,B 0,C 180,E1 -14143.677,E2 -14143.677} C_VEL
LIN {X 0,Y 343.018,Z 591.081,A -85,B 0,C 180,E1 -14145.448,E2 -14145.448} C_VEL
LIN {X 0,Y 344.943,Z 580.848,A -85,B 0,C 180,E1 -14147.184,E2 -14147.184} C_VEL
LIN {X 0,Y 346.929,Z 569.54,A -85,B 0,C 180,E1 -14148.76,E2 -14148.76} C_VEL
LIN {X 0,Y 348.126,Z 562.242,A -85,B 0,C 180,E1 -14149.611,E2 -14149.611} C_VEL
LIN {X 0,Y 348.445,Z 549.924,A -85,B 0,C 180,E1 -14150.973,E2 -14150.973} C_VEL
LIN {X 0,Y 347.397,Z 538.594,A -85,B 0,C 180,E1 -14152.168,E2 -14152.168} C_VEL
LIN {X 0,Y 345.322,Z 527.914,A -85,B 0,C 180,E1 -14153.268,E2 -14153.268} C_VEL
LIN {X 0,Y 342.047,Z 516.517,A -85,B 0,C 180,E1 -14154.486,E2 -14154.486} C_VEL
LIN {X 0,Y 340.936,Z 512.775,A -85,B 0,C 180,E1 -14154.86,E2 -14154.86} C_VEL
LIN {X 0,Y 340.89,Z 512.471,A -85,B 0,C 180,E1 -14154.888,E2 -14154.888} C_VEL
LIN {X 0,Y 341.816,Z 505.786,A -85,B 0,C 180,E1 -14158.894,E2 -14158.894} C_VEL
LIN {X 0,Y 342.723,Z 500.774,A -85,B 0,C 180,E1 -14162.22,E2 -14162.22} C_VEL
LIN {X 0,Y 343.565,Z 496.904,A -85,B 0,C 180,E1 -14165.091,E2 -14165.091} C_VEL
LIN {X 0,Y 343.924,Z 493.78,A -85,B 0,C 180,E1 -14167.81,E2 -14167.81} C_VEL
LIN {X 0,Y 343.664,Z 490.982,A -85,B 0,C 180,E1 -14170.875,E2 -14170.875} C_VEL
LIN {X 0,Y 343.335,Z 488.644,A -85,B 0,C 180,E1 -14174.238,E2 -14174.238} C_VEL
LIN {X 0,Y 343.009,Z 487.085,A -85,B 0,C 180,E1 -14177.529,E2 -14177.529} C_VEL
LIN {X 0,Y 342.739,Z 486.117,A -85,B 0,C 180,E1 -14181.188,E2 -14181.188} C_VEL
LIN {X 0,Y 342.592,Z 485.893,A -85,B 0,C 180,E1 -14183.494,E2 -14183.494} C_VEL
LIN {X 0,Y 342.085,Z 486.185,A -85,B 0,C 180,E1 -14187.388,E2 -14187.388} C_VEL
LIN {X 0,Y 341.651,Z 486.869,A -85,B 0,C 180,E1 -14190.416,E2 -14190.416} C_VEL
LIN {X 0,Y 341.106,Z 488.269,A -85,B 0,C 180,E1 -14194.363,E2 -14194.363} C_VEL
LIN {X 0,Y 341.043,Z 488.662,A -85,B 0,C 180,E1 -14195.293,E2 -14195.293} C_VEL
LIN {X 0,Y 341.671,Z 490.745,A -85,B 0,C 180,E1 -14195.533,E2 -14195.533} C_VEL
LIN {X 0,Y 344.946,Z 496.904,A -85,B 0,C 180,E1 -14196.469,E2 -14196.469} C_VEL
LIN {X 0,Y 349.037,Z 506.79,A -85,B 0,C 180,E1 -14197.855,E2 -14197.855} C_VEL
LIN {X 0,Y 351.653,Z 516.21,A -85,B 0,C 180,E1 -14199.095,E2 -14199.095} C_VEL
LIN {X 0,Y 352.15,Z 518.968,A -85,B 0,C 180,E1 -14199.449,E2 -14199.449} C_VEL
LIN {X 0,Y 350.123,Z 532.028,A -85,B 0,C 180,E1 -14200.827,E2 -14200.827} C_VEL
LIN {X 0,Y 348.413,Z 541.852,A -85,B 0,C 180,E1 -14202.118,E2 -14202.118} C_VEL
LIN {X 0,Y 346.41,Z 552.217,A -85,B 0,C 180,E1 -14203.802,E2 -14203.802} C_VEL
LIN {X 0,Y 344.986,Z 559.52,A -85,B 0,C 180,E1 -14205.247,E2 -14205.247} C_VEL
LIN {X 0,Y 343.489,Z 566.818,A -85,B 0,C 180,E1 -14206.993,E2 -14206.993} C_VEL
LIN {X 0,Y 342.385,Z 572.658,A -85,B 0,C 180,E1 -14208.755,E2 -14208.755} C_VEL
LIN {X 0,Y 341.397,Z 577.332,A -85,B 0,C 180,E1 -14210.521,E2 -14210.521} C_VEL
LIN {X 0,Y 340.811,Z 580.1,A -85,B 0,C 180,E1 -14211.823,E2 -14211.823} C_VEL
LIN {X 0,Y 340.325,Z 581.969,A -85,B 0,C 180,E1 -14212.883,E2 -14212.883} C_VEL
LIN {X 0,Y 340.031,Z 583.601,A -85,B 0,C 180,E1 -14214.069,E2 -14214.069} C_VEL
LIN {X 0,Y 339.966,Z 584.783,A -85,B 0,C 180,E1 -14215.257,E2 -14215.257} C_VEL
LIN {X 0,Y 339.738,Z 585.596,A -85,B 0,C 180,E1 -14216.442,E2 -14216.442} C_VEL
LIN {X 0,Y 339.542,Z 586.02,A -85,B 0,C 180,E1 -14217.628,E2 -14217.628} C_VEL
LIN {X 0,Y 339.404,Z 586.008,A -85,B 0,C 180,E1 -14218.814,E2 -14218.814} C_VEL
LIN {X 0,Y 339.34,Z 585.584,A -85,B 0,C 180,E1 -14220,E2 -14220} C_VEL
LIN {X 0,Y 339.328,Z 584.764,A -85,B 0,C 180,E1 -14221.187,E2 -14221.187} C_VEL
LIN {X 0,Y 339.331,Z 583.537,A -85,B 0,C 180,E1 -14222.374,E2 -14222.374} C_VEL
LIN {X 0,Y 339.395,Z 580.863,A -85,B 0,C 180,E1 -14224.157,E2 -14224.157} C_VEL
LIN {X 0,Y 339.642,Z 576.21,A -85,B 0,C 180,E1 -14226.32,E2 -14226.32} C_VEL
LIN {X 0,Y 340.017,Z 570.447,A -85,B 0,C 180,E1 -14228.319,E2 -14228.319} C_VEL
LIN {X 0,Y 340.568,Z 563.931,A -85,B 0,C 180,E1 -14230.103,E2 -14230.103} C_VEL
LIN {X 0,Y 341.218,Z 555.819,A -85,B 0,C 180,E1 -14231.887,E2 -14231.887} C_VEL
LIN {X 0,Y 342.131,Z 545.839,A -85,B 0,C 180,E1 -14233.665,E2 -14233.665} C_VEL
LIN {X 0,Y 343.114,Z 535.532,A -85,B 0,C 180,E1 -14235.139,E2 -14235.139} C_VEL
LIN {X 0,Y 343.995,Z 523.855,A -85,B 0,C 180,E1 -14236.497,E2 -14236.497} C_VEL
LIN {X 0,Y 344.747,Z 513.137,A -85,B 0,C 180,E1 -14237.5,E2 -14237.5} C_VEL
LIN {X 0,Y 345.031,Z 508.34,A -85,B 0,C 180,E1 -14237.884,E2 -14237.884} C_VEL
LIN {X 0,Y 342.242,Z 494.577,A -85,B 0,C 180,E1 -14238.919,E2 -14238.919} C_VEL
LIN {X 0,Y 339.505,Z 481.107,A -85,B 0,C 180,E1 -14239.697,E2 -14239.697} C_VEL
LIN {X 0,Y 339.53,Z 477.775,A -85,B 0,C 180,E1 -14243.16,E2 -14243.16} C_VEL
LIN {X 0,Y 339.735,Z 474.17,A -85,B 0,C 180,E1 -14247.072,E2 -14247.072} C_VEL
LIN {X 0,Y 340.041,Z 474.127,A -85,B 0,C 180,E1 -14249.765,E2 -14249.765} C_VEL
LIN {X 0,Y 340.298,Z 474.098,A -85,B 0,C 180,E1 -14252.478,E2 -14252.478} C_VEL
LIN {X 0,Y 340.557,Z 474.061,A -85,B 0,C 180,E1 -14255.299,E2 -14255.299} C_VEL
LIN {X 0,Y 340.707,Z 474.047,A -85,B 0,C 180,E1 -14258.385,E2 -14258.385} C_VEL
LIN {X 0,Y 340.703,Z 474.047,A -85,B 0,C 180,E1 -14262.046,E2 -14262.046} C_VEL
LIN {X 0,Y 340.656,Z 474.054,A -85,B 0,C 180,E1 -14266.227,E2 -14266.227} C_VEL
LIN {X 0,Y 340.693,Z 474.046,A -85,B 0,C 180,E1 -14269.753,E2 -14269.753} C_VEL
LIN {X 0,Y 340.71,Z 474.042,A -85,B 0,C 180,E1 -14273.259,E2 -14273.259} C_VEL
LIN {X 0,Y 340.699,Z 474.049,A -85,B 0,C 180,E1 -14276.154,E2 -14276.154} C_VEL
LIN {X 0,Y 340.746,Z 474.042,A -85,B 0,C 180,E1 -14280.329,E2 -14280.329} C_VEL
LIN {X 0,Y 340.808,Z 474.03,A -85,B 0,C 180,E1 -14283.02,E2 -14283.02} C_VEL
LIN {X 0,Y 340.761,Z 474.037,A -85,B 0,C 180,E1 -14285.638,E2 -14285.638} C_VEL
LIN {X 0,Y 340.753,Z 474.037,A -85,B 0,C 180,E1 -14289.474,E2 -14289.474} C_VEL
LIN {X 0,Y 340.863,Z 474.028,A -85,B 0,C 180,E1 -14291.984,E2 -14291.984} C_VEL
LIN {X 0,Y 340.874,Z 474.024,A -85,B 0,C 180,E1 -14295.705,E2 -14295.705} C_VEL
LIN {X 0,Y 340.875,Z 474.022,A -85,B 0,C 180,E1 -14299.306,E2 -14299.306} C_VEL
LIN {X 0,Y 341.061,Z 473.998,A -85,B 0,C 180,E1 -14302.898,E2 -14302.898} C_VEL
LIN {X 0,Y 341.173,Z 473.987,A -85,B 0,C 180,E1 -14307.639,E2 -14307.639} C_VEL
LIN {X 0,Y 341.3,Z 473.974,A -85,B 0,C 180,E1 -14310,E2 -14310} C_VEL
LIN {X 0,Y 341.173,Z 473.987,A -85,B 0,C 180,E1 -14312.361,E2 -14312.361} C_VEL
LIN {X 0,Y 341.023,Z 474.003,A -85,B 0,C 180,E1 -14317.103,E2 -14317.103} C_VEL
LIN {X 0,Y 340.876,Z 474.022,A -85,B 0,C 180,E1 -14320.693,E2 -14320.693} C_VEL
LIN {X 0,Y 340.867,Z 474.024,A -85,B 0,C 180,E1 -14324.324,E2 -14324.324} C_VEL
LIN {X 0,Y 340.842,Z 474.027,A -85,B 0,C 180,E1 -14328.467,E2 -14328.467} C_VEL
LIN {X 0,Y 340.757,Z 474.042,A -85,B 0,C 180,E1 -14331.856,E2 -14331.856} C_VEL
LIN {X 0,Y 340.776,Z 474.038,A -85,B 0,C 180,E1 -14335.664,E2 -14335.664} C_VEL
LIN {X 0,Y 340.732,Z 474.041,A -85,B 0,C 180,E1 -14338.32,E2 -14338.32} C_VEL
LIN {X 0,Y 340.701,Z 474.043,A -85,B 0,C 180,E1 -14341.044,E2 -14341.044} C_VEL
LIN {X 0,Y 340.722,Z 474.042,A -85,B 0,C 180,E1 -14345.278,E2 -14345.278} C_VEL
LIN {X 0,Y 340.715,Z 474.042,A -85,B 0,C 180,E1 -14348.386,E2 -14348.386} C_VEL
LIN {X 0,Y 340.701,Z 474.046,A -85,B 0,C 180,E1 -14352.045,E2 -14352.045} C_VEL
LIN {X 0,Y 340.654,Z 474.05,A -85,B 0,C 180,E1 -14356.226,E2 -14356.226} C_VEL
LIN {X 0,Y 340.691,Z 474.05,A -85,B 0,C 180,E1 -14359.752,E2 -14359.752} C_VEL
LIN {X 0,Y 340.707,Z 474.044,A -85,B 0,C 180,E1 -14363.258,E2 -14363.258} C_VEL
LIN {X 0,Y 340.695,Z 474.045,A -85,B 0,C 180,E1 -14366.153,E2 -14366.153} C_VEL
LIN {X 0,Y 340.776,Z 474.034,A -85,B 0,C 180,E1 -14370.332,E2 -14370.332} C_VEL
LIN {X 0,Y 340.748,Z 474.037,A -85,B 0,C 180,E1 -14370.692,E2 -14370.692} C_VEL
LIN {X 0,Y 340.051,Z 474.129,A -85,B 0,C 180,E1 -14371.679,E2 -14371.679} C_VEL
LIN {X 0,Y 337.197,Z 474.482,A -85,B 0,C 180,E1 -14373.284,E2 -14373.284} C_VEL
LIN {X 0,Y 334.795,Z 474.778,A -85,B 0,C 180,E1 -14374.584,E2 -14374.584} C_VEL
LIN {X 0,Y 333.761,Z 474.913,A -85,B 0,C 180,E1 -14375.59,E2 -14375.59} C_VEL
LIN {X 0,Y 333.674,Z 474.916,A -85,B 0,C 180,E1 -14375.931,E2 -14375.931} C_VEL
LIN {X 0,Y 333.683,Z 474.918,A -85,B 0,C 180,E1 -14379.019,E2 -14379.019} C_VEL
LIN {X 0,Y 333.796,Z 474.909,A -85,B 0,C 180,E1 -14381.589,E2 -14381.589} C_VEL
LIN {X 0,Y 333.809,Z 474.907,A -85,B 0,C 180,E1 -14385.576,E2 -14385.576} C_VEL
LIN {X 0,Y 333.835,Z 474.9,A -85,B 0,C 180,E1 -14389.078,E2 -14389.078} C_VEL
LIN {X 0,Y 334.026,Z 474.875,A -85,B 0,C 180,E1 -14392.747,E2 -14392.747} C_VEL
LIN {X 0,Y 333.811,Z 474.903,A -85,B 0,C 180,E1 -14395.169,E2 -14395.169} C_VEL
LIN {X 0,Y 334.107,Z 474.869,A -85,B 0,C 180,E1 -14397.589,E2 -14397.589} C_VEL
LIN {X 0,Y 334.248,Z 474.848,A -85,B 0,C 180,E1 -14400,E2 -14400} C_VEL
LIN {X 0,Y 334.106,Z 474.864,A -85,B 0,C 180,E1 -14402.411,E2 -14402.411} C_VEL
LIN {X 0,Y 334.026,Z 474.878,A -85,B 0,C 180,E1 -14407.252,E2 -14407.252} C_VEL
LIN {X 0,Y 333.834,Z 474.899,A -85,B 0,C 180,E1 -14410.922,E2 -14410.922} C_VEL
LIN {X 0,Y 333.808,Z 474.902,A -85,B 0,C 180,E1 -14414.634,E2 -14414.634} C_VEL
LIN {X 0,Y 333.796,Z 474.903,A -85,B 0,C 180,E1 -14418.655,E2 -14418.655} C_VEL
LIN {X 0,Y 333.692,Z 474.916,A -85,B 0,C 180,E1 -14422.278,E2 -14422.278} C_VEL
LIN {X 0,Y 333.735,Z 474.911,A -85,B 0,C 180,E1 -14426.246,E2 -14426.246} C_VEL
LIN {X 0,Y 333.69,Z 474.919,A -85,B 0,C 180,E1 -14428.974,E2 -14428.974} C_VEL
LIN {X 0,Y 333.645,Z 474.922,A -85,B 0,C 180,E1 -14432.588,E2 -14432.588} C_VEL
LIN {X 0,Y 333.677,Z 474.918,A -85,B 0,C 180,E1 -14436.139,E2 -14436.139} C_VEL
LIN {X 0,Y 333.682,Z 474.922,A -85,B 0,C 180,E1 -14439.187,E2 -14439.187} C_VEL
LIN {X 0,Y 333.689,Z 474.917,A -85,B 0,C 180,E1 -14442.511,E2 -14442.511} C_VEL
LIN {X 0,Y 333.734,Z 474.922,A -85,B 0,C 180,E1 -14444.746,E2 -14444.746} C_VEL
LIN {X 0,Y 334.903,Z 481.559,A -85,B 0,C 180,E1 -14449.066,E2 -14449.066} C_VEL
LIN {X 0,Y 335.854,Z 487.407,A -85,B 0,C 180,E1 -14452.672,E2 -14452.672} C_VEL
LIN {X 0,Y 335.789,Z 490.904,A -85,B 0,C 180,E1 -14454.712,E2 -14454.712} C_VEL
LIN {X 0,Y 335.089,Z 496.145,A -85,B 0,C 180,E1 -14457.668,E2 -14457.668} C_VEL
LIN {X 0,Y 334.352,Z 502.334,A -85,B 0,C 180,E1 -14461.089,E2 -14461.089} C_VEL
LIN {X 0,Y 333.53,Z 509.702,A -85,B 0,C 180,E1 -14465.075,E2 -14465.075} C_VEL
LIN {X 0,Y 332.826,Z 518.193,A -85,B 0,C 180,E1 -14469.61,E2 -14469.61} C_VEL
LIN {X 0,Y 332.788,Z 518.8,A -85,B 0,C 180,E1 -14469.93,E2 -14469.93} C_VEL
LIN {X 0,Y 334.308,Z 532.723,A -85,B 0,C 180,E1 -14470.651,E2 -14470.651} C_VEL
LIN {X 0,Y 335.9,Z 546.474,A -85,B 0,C 180,E1 -14471.626,E2 -14471.626} C_VEL
LIN {X 0,Y 336.807,Z 556.89,A -85,B 0,C 180,E1 -14472.545,E2 -14472.545} C_VEL
LIN {X 0,Y 335.937,Z 568.432,A -85,B 0,C 180,E1 -14473.751,E2 -14473.751} C_VEL
LIN {X 0,Y 334.764,Z 579.627,A -85,B 0,C 180,E1 -14475.218,E2 -14475.218} C_VEL
LIN {X 0,Y 333.994,Z 588.374,A -85,B 0,C 180,E1 -14476.617,E2 -14476.617} C_VEL
LIN {X 0,Y 333.343,Z 596.289,A -85,B 0,C 180,E1 -14478.138,E2 -14478.138} C_VEL
LIN {X 0,Y 332.769,Z 604.074,A -85,B 0,C 180,E1 -14479.966,E2 -14479.966} C_VEL
LIN {X 0,Y 332.361,Z 611.206,A -85,B 0,C 180,E1 -14482.1,E2 -14482.1} C_VEL
LIN {X 0,Y 332.18,Z 615.928,A -85,B 0,C 180,E1 -14483.928,E2 -14483.928} C_VEL
LIN {X 0,Y 332.237,Z 618.441,A -85,B 0,C 180,E1 -14485.146,E2 -14485.146} C_VEL
LIN {X 0,Y 332.117,Z 620.412,A -85,B 0,C 180,E1 -14486.36,E2 -14486.36} C_VEL
LIN {X 0,Y 332.215,Z 621.966,A -85,B 0,C 180,E1 -14487.575,E2 -14487.575} C_VEL
LIN {X 0,Y 332.293,Z 623.081,A -85,B 0,C 180,E1 -14488.788,E2 -14488.788} C_VEL
LIN {X 0,Y 332.277,Z 623.714,A -85,B 0,C 180,E1 -14490,E2 -14490} C_VEL
LIN {X 0,Y 332.252,Z 623.93,A -85,B 0,C 180,E1 -14491.212,E2 -14491.212} C_VEL
LIN {X 0,Y 332.081,Z 623.725,A -85,B 0,C 180,E1 -14492.426,E2 -14492.426} C_VEL
LIN {X 0,Y 332.058,Z 623.108,A -85,B 0,C 180,E1 -14493.641,E2 -14493.641} C_VEL
LIN {X 0,Y 332.045,Z 620.869,A -85,B 0,C 180,E1 -14495.849,E2 -14495.849} C_VEL
LIN {X 0,Y 332.321,Z 617.551,A -85,B 0,C 180,E1 -14497.901,E2 -14497.901} C_VEL
LIN {X 0,Y 332.748,Z 613.523,A -85,B 0,C 180,E1 -14499.728,E2 -14499.728} C_VEL
LIN {X 0,Y 333.403,Z 608.444,A -85,B 0,C 180,E1 -14501.552,E2 -14501.552} C_VEL
LIN {X 0,Y 334.728,Z 601.004,A -85,B 0,C 180,E1 -14503.663,E2 -14503.663} C_VEL
LIN {X 0,Y 335.98,Z 593.085,A -85,B 0,C 180,E1 -14505.468,E2 -14505.468} C_VEL
LIN {X 0,Y 337.854,Z 583.555,A -85,B 0,C 180,E1 -14507.243,E2 -14507.243} C_VEL
LIN {X 0,Y 339.885,Z 572.985,A -85,B 0,C 180,E1 -14508.85,E2 -14508.85} C_VEL
LIN {X 0,Y 341.693,Z 562.536,A -85,B 0,C 180,E1 -14510.153,E2 -14510.153} C_VEL
LIN {X 0,Y 342.125,Z 551.12,A -85,B 0,C 180,E1 -14511.491,E2 -14511.491} C_VEL
LIN {X 0,Y 341.158,Z 539.752,A -85,B 0,C 180,E1 -14512.758,E2 -14512.758} C_VEL
LIN {X 0,Y 339.074,Z 528.888,A -85,B 0,C 180,E1 -14513.987,E2 -14513.987} C_VEL
LIN {X 0,Y 335.758,Z 516.939,A -85,B 0,C 180,E1 -14515.361,E2 -14515.361} C_VEL
LIN {X 0,Y 334.241,Z 512.747,A -85,B 0,C 180,E1 -14515.872,E2 -14515.872} C_VEL
LIN {X 0,Y 334.082,Z 511.612,A -85,B 0,C 180,E1 -14516.01,E2 -14516.01} C_VEL
LIN {X 0,Y 334.959,Z 505.999,A -85,B 0,C 180,E1 -14519.543,E2 -14519.543} C_VEL
LIN {X 0,Y 336.045,Z 500.735,A -85,B 0,C 180,E1 -14523.222,E2 -14523.222} C_VEL
LIN {X 0,Y 336.708,Z 497.527,A -85,B 0,C 180,E1 -14525.764,E2 -14525.764} C_VEL
LIN {X 0,Y 336.986,Z 495.504,A -85,B 0,C 180,E1 -14527.58,E2 -14527.58} C_VEL
LIN {X 0,Y 336.772,Z 492.993,A -85,B 0,C 180,E1 -14530.311,E2 -14530.311} C_VEL
LIN {X 0,Y 336.457,Z 490.624,A -85,B 0,C 180,E1 -14533.576,E2 -14533.576} C_VEL
LIN {X 0,Y 336.131,Z 488.849,A -85,B 0,C 180,E1 -14537.038,E2 -14537.038} C_VEL
LIN {X 0,Y 335.844,Z 487.754,A -85,B 0,C 180,E1 -14540.74,E2 -14540.74} C_VEL
LIN {X 0,Y 335.564,Z 487.416,A -85,B 0,C 180,E1 -14544.096,E2 -14544.096} C_VEL
LIN {X 0,Y 335.192,Z 487.593,A -85,B 0,C 180,E1 -14547.002,E2 -14547.002} C_VEL
LIN {X 0,Y 334.82,Z 488.108,A -85,B 0,C 180,E1 -14549.75,E2 -14549.75} C_VEL
LIN {X 0,Y 334.374,Z 488.911,A -85,B 0,C 180,E1 -14552.458,E2 -14552.458} C_VEL
LIN {X 0,Y 334.191,Z 489.752,A -85,B 0,C 180,E1 -14554.235,E2 -14554.235} C_VEL
LIN {X 0,Y 334.841,Z 491.695,A -85,B 0,C 180,E1 -14554.493,E2 -14554.493} C_VEL
LIN {X 0,Y 336.56,Z 494.565,A -85,B 0,C 180,E1 -14555,E2 -14555} C_VEL
LIN {X 0,Y 341.644,Z 505.532,A -85,B 0,C 180,E1 -14556.726,E2 -14556.726} C_VEL
LIN {X 0,Y 344.432,Z 513.763,A -85,B 0,C 180,E1 -14557.939,E2 -14557.939} C_VEL
LIN {X 0,Y 345.963,Z 520.423,A -85,B 0,C 180,E1 -14558.865,E2 -14558.865} C_VEL
LIN {X 0,Y 344.075,Z 532.638,A -85,B 0,C 180,E1 -14560.219,E2 -14560.219} C_VEL
LIN {X 0,Y 342.322,Z 541.786,A -85,B 0,C 180,E1 -14561.445,E2 -14561.445} C_VEL
LIN {X 0,Y 340.466,Z 550.839,A -85,B 0,C 180,E1 -14562.893,E2 -14562.893} C_VEL
LIN {X 0,Y 338.779,Z 558.414,A -85,B 0,C 180,E1 -14564.355,E2 -14564.355} C_VEL
LIN {X 0,Y 336.946,Z 567.019,A -85,B 0,C 180,E1 -14566.429,E2 -14566.429} C_VEL
LIN {X 0,Y 335.512,Z 573.784,A -85,B 0,C 180,E1 -14568.522,E2 -14568.522} C_VEL
LIN {X 0,Y 334.466,Z 578.325,A -85,B 0,C 180,E1 -14570.323,E2 -14570.323} C_VEL
LIN {X 0,Y 333.85,Z 581.013,A -85,B 0,C 180,E1 -14571.659,E2 -14571.659} C_VEL
LIN {X 0,Y 333.328,Z 582.772,A -85,B 0,C 180,E1 -14572.733,E2 -14572.733} C_VEL
LIN {X 0,Y 332.997,Z 584.305,A -85,B 0,C 180,E1 -14573.943,E2 -14573.943} C_VEL
LIN {X 0,Y 332.933,Z 585.431,A -85,B 0,C 180,E1 -14575.157,E2 -14575.157} C_VEL
LIN {X 0,Y 332.7,Z 586.188,A -85,B 0,C 180,E1 -14576.367,E2 -14576.367} C_VEL
LIN {X 0,Y 332.491,Z 586.523,A -85,B 0,C 180,E1 -14577.577,E2 -14577.577} C_VEL
LIN {X 0,Y 332.346,Z 586.435,A -85,B 0,C 180,E1 -14578.789,E2 -14578.789} C_VEL
LIN {X 0,Y 332.262,Z 585.954,A -85,B 0,C 180,E1 -14580,E2 -14580} C_VEL
LIN {X 0,Y 332.236,Z 585.078,A -85,B 0,C 180,E1 -14581.212,E2 -14581.212} C_VEL
LIN {X 0,Y 332.235,Z 583.755,A -85,B 0,C 180,E1 -14582.425,E2 -14582.425} C_VEL
LIN {X 0,Y 332.329,Z 580.982,A -85,B 0,C 180,E1 -14584.245,E2 -14584.245} C_VEL
LIN {X 0,Y 332.529,Z 577.163,A -85,B 0,C 180,E1 -14586.066,E2 -14586.066} C_VEL
LIN {X 0,Y 332.844,Z 572.204,A -85,B 0,C 180,E1 -14587.889,E2 -14587.889} C_VEL
LIN {X 0,Y 333.429,Z 564.814,A -85,B 0,C 180,E1 -14590.015,E2 -14590.015} C_VEL
LIN {X 0,Y 334.107,Z 556.824,A -85,B 0,C 180,E1 -14591.835,E2 -14591.835} C_VEL
LIN {X 0,Y 335.012,Z 546.946,A -85,B 0,C 180,E1 -14593.651,E2 -14593.651} C_VEL
LIN {X 0,Y 335.997,Z 536.831,A -85,B 0,C 180,E1 -14595.157,E2 -14595.157} C_VEL
LIN {X 0,Y 336.893,Z 525.046,A -85,B 0,C 180,E1 -14596.579,E2 -14596.579} C_VEL
LIN {X 0,Y 337.777,Z 513.254,A -85,B 0,C 180,E1 -14597.716,E2 -14597.716} C_VEL
LIN {X 0,Y 337.942,Z 508.651,A -85,B 0,C 180,E1 -14598.099,E2 -14598.099} C_VEL
LIN {X 0,Y 335.191,Z 495.353,A -85,B 0,C 180,E1 -14599.12,E2 -14599.12} C_VEL
LIN {X 0,Y 332.43,Z 481.496,A -85,B 0,C 180,E1 -14599.932,E2 -14599.932} C_VEL
LIN {X 0,Y 332.467,Z 477.936,A -85,B 0,C 180,E1 -14603.681,E2 -14603.681} C_VEL
LIN {X 0,Y 332.597,Z 475.453,A -85,B 0,C 180,E1 -14606.343,E2 -14606.343} C_VEL
LIN {X 0,Y 332.737,Z 475.042,A -85,B 0,C 180,E1 -14607.69,E2 -14607.69} C_VEL
LIN {X 0,Y 333.033,Z 475.003,A -85,B 0,C 180,E1 -14610.43,E2 -14610.43} C_VEL
LIN {X 0,Y 333.306,Z 474.964,A -85,B 0,C 180,E1 -14613.246,E2 -14613.246} C_VEL
LIN {X 0,Y 333.635,Z 474.924,A -85,B 0,C 180,E1 -14616.825,E2 -14616.825} C_VEL
LIN {X 0,Y 333.651,Z 474.923,A -85,B 0,C 180,E1 -14620.685,E2 -14620.685} C_VEL
LIN {X 0,Y 333.598,Z 474.933,A -85,B 0,C 180,E1 -14624.251,E2 -14624.251} C_VEL
LIN {X 0,Y 333.646,Z 474.922,A -85,B 0,C 180,E1 -14627.619,E2 -14627.619} C_VEL
LIN {X 0,Y 333.657,Z 474.92,A -85,B 0,C 180,E1 -14631.202,E2 -14631.202} C_VEL
LIN {X 0,Y 333.681,Z 474.92,A -85,B 0,C 180,E1 -14633.861,E2 -14633.861} C_VEL
LIN {X 0,Y 333.65,Z 474.921,A -85,B 0,C 180,E1 -14637.412,E2 -14637.412} C_VEL
LIN {X 0,Y 333.695,Z 474.915,A -85,B 0,C 180,E1 -14641.026,E2 -14641.026} C_VEL
LIN {X 0,Y 333.74,Z 474.912,A -85,B 0,C 180,E1 -14643.754,E2 -14643.754} C_VEL
LIN {X 0,Y 333.724,Z 474.916,A -85,B 0,C 180,E1 -14647.914,E2 -14647.914} C_VEL
LIN {X 0,Y 333.8,Z 474.904,A -85,B 0,C 180,E1 -14651.589,E2 -14651.589} C_VEL
LIN {X 0,Y 333.813,Z 474.902,A -85,B 0,C 180,E1 -14655.576,E2 -14655.576} C_VEL
LIN {X 0,Y 333.838,Z 474.898,A -85,B 0,C 180,E1 -14659.078,E2 -14659.078} C_VEL
LIN {X 0,Y 334.009,Z 474.877,A -85,B 0,C 180,E1 -14662.747,E2 -14662.747} C_VEL
LIN {X 0,Y 333.813,Z 474.901,A -85,B 0,C 180,E1 -14665.169,E2 -14665.169} C_VEL
LIN {X 0,Y 334.11,Z 474.866,A -85,B 0,C 180,E1 -14667.589,E2 -14667.589} C_VEL
LIN {X 0,Y 334.251,Z 474.852,A -85,B 0,C 180,E1 -14670,E2 -14670} C_VEL
LIN {X 0,Y 334.11,Z 474.866,A -85,B 0,C 180,E1 -14672.411,E2 -14672.411} C_VEL
LIN {X 0,Y 334.006,Z 474.882,A -85,B 0,C 180,E1 -14676.039,E2 -14676.039} C_VEL
LIN {X 0,Y 333.854,Z 474.899,A -85,B 0,C 180,E1 -14679.695,E2 -14679.695} C_VEL
LIN {X 0,Y 333.801,Z 474.903,A -85,B 0,C 180,E1 -14683.391,E2 -14683.391} C_VEL
LIN {X 0,Y 333.751,Z 474.909,A -85,B 0,C 180,E1 -14687.146,E2 -14687.146} C_VEL
LIN {X 0,Y 333.743,Z 474.913,A -85,B 0,C 180,E1 -14689.69,E2 -14689.69} C_VEL
LIN {X 0,Y 333.696,Z 474.918,A -85,B 0,C 180,E1 -14692.278,E2 -14692.278} C_VEL
LIN {X 0,Y 333.739,Z 474.912,A -85,B 0,C 180,E1 -14696.246,E2 -14696.246} C_VEL
LIN {X 0,Y 333.693,Z 474.916,A -85,B 0,C 180,E1 -14698.974,E2 -14698.974} C_VEL
LIN {X 0,Y 333.649,Z 474.922,A -85,B 0,C 180,E1 -14702.587,E2 -14702.587} C_VEL
LIN {X 0,Y 333.68,Z 474.92,A -85,B 0,C 180,E1 -14706.138,E2 -14706.138} C_VEL
LIN {X 0,Y 333.65,Z 474.922,A -85,B 0,C 180,E1 -14709.192,E2 -14709.192} C_VEL
LIN {X 0,Y 333.635,Z 474.923,A -85,B 0,C 180,E1 -14712.5,E2 -14712.5} C_VEL
LIN {X 0,Y 333.599,Z 474.931,A -85,B 0,C 180,E1 -14715.955,E2 -14715.955} C_VEL
LIN {X 0,Y 333.649,Z 474.923,A -85,B 0,C 180,E1 -14719.315,E2 -14719.315} C_VEL
LIN {X 0,Y 333.667,Z 474.92,A -85,B 0,C 180,E1 -14723.167,E2 -14723.167} C_VEL
LIN {X 0,Y 333.64,Z 474.922,A -85,B 0,C 180,E1 -14726.791,E2 -14726.791} C_VEL
LIN {X 0,Y 333.694,Z 474.916,A -85,B 0,C 180,E1 -14730.7,E2 -14730.7} C_VEL
LIN {X 0,Y 333.737,Z 474.915,A -85,B 0,C 180,E1 -14733.753,E2 -14733.753} C_VEL
LIN {X 0,Y 333.674,Z 474.916,A -85,B 0,C 180,E1 -14735.931,E2 -14735.931} C_VEL
LIN {X 0,Y 333.024,Z 475,A -85,B 0,C 180,E1 -14736.937,E2 -14736.937} C_VEL
LIN {X 0,Y 330.261,Z 475.351,A -85,B 0,C 180,E1 -14738.577,E2 -14738.577} C_VEL
LIN {X 0,Y 327.895,Z 475.646,A -85,B 0,C 180,E1 -14739.905,E2 -14739.905} C_VEL
LIN {X 0,Y 326.842,Z 475.773,A -85,B 0,C 180,E1 -14740.931,E2 -14740.931} C_VEL
LIN {X 0,Y 326.736,Z 475.783,A -85,B 0,C 180,E1 -14741.279,E2 -14741.279} C_VEL
LIN {X 0,Y 326.764,Z 475.783,A -85,B 0,C 180,E1 -14745.433,E2 -14745.433} C_VEL
LIN {X 0,Y 326.771,Z 475.778,A -85,B 0,C 180,E1 -14748.839,E2 -14748.839} C_VEL
LIN {X 0,Y 326.98,Z 475.752,A -85,B 0,C 180,E1 -14752.59,E2 -14752.59} C_VEL
LIN {X 0,Y 326.778,Z 475.779,A -85,B 0,C 180,E1 -14755.065,E2 -14755.065} C_VEL
LIN {X 0,Y 327.048,Z 475.749,A -85,B 0,C 180,E1 -14757.536,E2 -14757.536} C_VEL
LIN {X 0,Y 327.199,Z 475.726,A -85,B 0,C 180,E1 -14760,E2 -14760} C_VEL
LIN {X 0,Y 327.047,Z 475.743,A -85,B 0,C 180,E1 -14762.463,E2 -14762.463} C_VEL
LIN {X 0,Y 326.997,Z 475.75,A -85,B 0,C 180,E1 -14766.169,E2 -14766.169} C_VEL
LIN {X 0,Y 326.915,Z 475.76,A -85,B 0,C 180,E1 -14768.655,E2 -14768.655} C_VEL
LIN {X 0,Y 326.734,Z 475.782,A -85,B 0,C 180,E1 -14772.421,E2 -14772.421} C_VEL
LIN {X 0,Y 326.754,Z 475.782,A -85,B 0,C 180,E1 -14774.957,E2 -14774.957} C_VEL
LIN {X 0,Y 326.732,Z 475.784,A -85,B 0,C 180,E1 -14778.838,E2 -14778.838} C_VEL
LIN {X 0,Y 326.621,Z 475.798,A -85,B 0,C 180,E1 -14782.787,E2 -14782.787} C_VEL
LIN {X 0,Y 326.69,Z 475.793,A -85,B 0,C 180,E1 -14785.484,E2 -14785.484} C_VEL
LIN {X 0,Y 326.647,Z 475.796,A -85,B 0,C 180,E1 -14789.66,E2 -14789.66} C_VEL
LIN {X 0,Y 326.618,Z 475.799,A -85,B 0,C 180,E1 -14792.947,E2 -14792.947} C_VEL
LIN {X 0,Y 326.613,Z 475.801,A -85,B 0,C 180,E1 -14795.519,E2 -14795.519} C_VEL
LIN {X 0,Y 326.643,Z 475.799,A -85,B 0,C 180,E1 -14799.234,E2 -14799.234} C_VEL
LIN {X 0,Y 326.634,Z 475.798,A -85,B 0,C 180,E1 -14802.983,E2 -14802.983} C_VEL
LIN {X 0,Y 326.719,Z 475.984,A -85,B 0,C 180,E1 -14804.669,E2 -14804.669} C_VEL
LIN {X 0,Y 327.753,Z 481.929,A -85,B 0,C 180,E1 -14808.634,E2 -14808.634} C_VEL
LIN {X 0,Y 328.733,Z 487.689,A -85,B 0,C 180,E1 -14812.281,E2 -14812.281} C_VEL
LIN {X 0,Y 328.801,Z 491.054,A -85,B 0,C 180,E1 -14814.315,E2 -14814.315} C_VEL
LIN {X 0,Y 328.33,Z 494.992,A -85,B 0,C 180,E1 -14816.596,E2 -14816.596} C_VEL
LIN {X 0,Y 327.433,Z 501.712,A -85,B 0,C 180,E1 -14820.418,E2 -14820.418} C_VEL
LIN {X 0,Y 326.549,Z 509.054,A -85,B 0,C 180,E1 -14824.505,E2 -14824.505} C_VEL
LIN {X 0,Y 325.867,Z 516.31,A -85,B 0,C 180,E1 -14828.492,E2 -14828.492} C_VEL
LIN {X 0,Y 325.74,Z 518.641,A -85,B 0,C 180,E1 -14829.682,E2 -14829.682} C_VEL
LIN {X 0,Y 327.105,Z 531.497,A -85,B 0,C 180,E1 -14830.355,E2 -14830.355} C_VEL
LIN {X 0,Y 328.553,Z 544.63,A -85,B 0,C 180,E1 -14831.285,E2 -14831.285} C_VEL
LIN {X 0,Y 329.668,Z 556.147,A -85,B 0,C 180,E1 -14832.315,E2 -14832.315} C_VEL
LIN {X 0,Y 329.39,Z 562.312,A -85,B 0,C 180,E1 -14832.94,E2 -14832.94} C_VEL
LIN {X 0,Y 328.401,Z 572.956,A -85,B 0,C 180,E1 -14834.202,E2 -14834.202} C_VEL
LIN {X 0,Y 327.457,Z 583.252,A -85,B 0,C 180,E1 -14835.711,E2 -14835.711} C_VEL
LIN {X 0,Y 326.637,Z 591.937,A -85,B 0,C 180,E1 -14837.259,E2 -14837.259} C_VEL
LIN {X 0,Y 325.855,Z 600.465,A -85,B 0,C 180,E1 -14839.122,E2 -14839.122} C_VEL
LIN {X 0,Y 325.466,Z 607.32,A -85,B 0,C 180,E1 -14840.993,E2 -14840.993} C_VEL
LIN {X 0,Y 325.179,Z 613.591,A -85,B 0,C 180,E1 -14843.173,E2 -14843.173} C_VEL
LIN {X 0,Y 325.172,Z 617.645,A -85,B 0,C 180,E1 -14845.041,E2 -14845.041} C_VEL
LIN {X 0,Y 325.047,Z 619.694,A -85,B 0,C 180,E1 -14846.281,E2 -14846.281} C_VEL
LIN {X 0,Y 325.128,Z 621.296,A -85,B 0,C 180,E1 -14847.522,E2 -14847.522} C_VEL
LIN {X 0,Y 325.233,Z 622.469,A -85,B 0,C 180,E1 -14848.762,E2 -14848.762} C_VEL
LIN {X 0,Y 325.219,Z 623.191,A -85,B 0,C 180,E1 -14850,E2 -14850} C_VEL
LIN {X 0,Y 325.17,Z 623.453,A -85,B 0,C 180,E1 -14851.239,E2 -14851.239} C_VEL
LIN {X 0,Y 324.98,Z 622.741,A -85,B 0,C 180,E1 -14853.72,E2 -14853.72} C_VEL
LIN {X 0,Y 324.962,Z 620.843,A -85,B 0,C 180,E1 -14855.818,E2 -14855.818} C_VEL
LIN {X 0,Y 325.252,Z 617.448,A -85,B 0,C 180,E1 -14858.074,E2 -14858.074} C_VEL
LIN {X 0,Y 325.737,Z 613.565,A -85,B 0,C 180,E1 -14859.94,E2 -14859.94} C_VEL
LIN {X 0,Y 326.42,Z 608.608,A -85,B 0,C 180,E1 -14861.803,E2 -14861.803} C_VEL
LIN {X 0,Y 327.844,Z 601.329,A -85,B 0,C 180,E1 -14863.956,E2 -14863.956} C_VEL
LIN {X 0,Y 329.16,Z 593.753,A -85,B 0,C 180,E1 -14865.788,E2 -14865.788} C_VEL
LIN {X 0,Y 331.145,Z 584.429,A -85,B 0,C 180,E1 -14867.604,E2 -14867.604} C_VEL
LIN {X 0,Y 333.499,Z 573.191,A -85,B 0,C 180,E1 -14869.385,E2 -14869.385} C_VEL
LIN {X 0,Y 335.238,Z 564.279,A -85,B 0,C 180,E1 -14870.558,E2 -14870.558} C_VEL
LIN {X 0,Y 335.872,Z 553.141,A -85,B 0,C 180,E1 -14871.934,E2 -14871.934} C_VEL
LIN {X 0,Y 335.071,Z 541.553,A -85,B 0,C 180,E1 -14873.329,E2 -14873.329} C_VEL
LIN {X 0,Y 332.85,Z 529.575,A -85,B 0,C 180,E1 -14874.779,E2 -14874.779} C_VEL
LIN {X 0,Y 330.498,Z 520.617,A -85,B 0,C 180,E1 -14875.895,E2 -14875.895} C_VEL
LIN {X 0,Y 328.335,Z 514.561,A -85,B 0,C 180,E1 -14876.726,E2 -14876.726} C_VEL
LIN {X 0,Y 327.337,Z 510.823,A -85,B 0,C 180,E1 -14877.188,E2 -14877.188} C_VEL
LIN {X 0,Y 328.423,Z 504.938,A -85,B 0,C 180,E1 -14881.133,E2 -14881.133} C_VEL
LIN {X 0,Y 329.194,Z 501.458,A -85,B 0,C 180,E1 -14883.716,E2 -14883.716} C_VEL
LIN {X 0,Y 329.893,Z 498.012,A -85,B 0,C 180,E1 -14886.621,E2 -14886.621} C_VEL
LIN {X 0,Y 330.01,Z 496.447,A -85,B 0,C 180,E1 -14888.141,E2 -14888.141} C_VEL
LIN {X 0,Y 329.892,Z 494.848,A -85,B 0,C 180,E1 -14889.92,E2 -14889.92} C_VEL
LIN {X 0,Y 329.559,Z 492.228,A -85,B 0,C 180,E1 -14893.526,E2 -14893.526} C_VEL
LIN {X 0,Y 329.222,Z 490.494,A -85,B 0,C 180,E1 -14896.913,E2 -14896.913} C_VEL
LIN {X 0,Y 328.934,Z 489.424,A -85,B 0,C 180,E1 -14900.28,E2 -14900.28} C_VEL
LIN {X 0,Y 328.705,Z 488.991,A -85,B 0,C 180,E1 -14903.226,E2 -14903.226} C_VEL
LIN {X 0,Y 328.307,Z 489.046,A -85,B 0,C 180,E1 -14906.602,E2 -14906.602} C_VEL
LIN {X 0,Y 327.951,Z 489.407,A -85,B 0,C 180,E1 -14909.048,E2 -14909.048} C_VEL
LIN {X 0,Y 327.317,Z 490.485,A -85,B 0,C 180,E1 -14913.005,E2 -14913.005} C_VEL
LIN {X 0,Y 327.849,Z 492.242,A -85,B 0,C 180,E1 -14913.246,E2 -14913.246} C_VEL
LIN {X 0,Y 329.801,Z 495.19,A -85,B 0,C 180,E1 -14913.864,E2 -14913.864} C_VEL
LIN {X 0,Y 334.993,Z 506.267,A -85,B 0,C 180,E1 -14915.786,E2 -14915.786} C_VEL
LIN {X 0,Y 338.442,Z 516.1,A -85,B 0,C 180,E1 -14917.358,E2 -14917.358} C_VEL
LIN {X 0,Y 339.828,Z 522.457,A -85,B 0,C 180,E1 -14918.32,E2 -14918.32} C_VEL
LIN {X 0,Y 339.407,Z 526.222,A -85,B 0,C 180,E1 -14918.754,E2 -14918.754} C_VEL
LIN {X 0,Y 337.032,Z 538.427,A -85,B 0,C 180,E1 -14920.241,E2 -14920.241} C_VEL
LIN {X 0,Y 334.655,Z 549.468,A -85,B 0,C 180,E1 -14921.955,E2 -14921.955} C_VEL
LIN {X 0,Y 332.423,Z 558.704,A -85,B 0,C 180,E1 -14923.732,E2 -14923.732} C_VEL
LIN {X 0,Y 330.682,Z 566.235,A -85,B 0,C 180,E1 -14925.539,E2 -14925.539} C_VEL
LIN {X 0,Y 329.09,Z 573.262,A -85,B 0,C 180,E1 -14927.669,E2 -14927.669} C_VEL
LIN {X 0,Y 327.864,Z 578,A -85,B 0,C 180,E1 -14929.502,E2 -14929.502} C_VEL
LIN {X 0,Y 326.901,Z 581.902,A -85,B 0,C 180,E1 -14931.476,E2 -14931.476} C_VEL
LIN {X 0,Y 326.335,Z 583.585,A -85,B 0,C 180,E1 -14932.576,E2 -14932.576} C_VEL
LIN {X 0,Y 325.97,Z 585.047,A -85,B 0,C 180,E1 -14933.812,E2 -14933.812} C_VEL
LIN {X 0,Y 325.902,Z 586.094,A -85,B 0,C 180,E1 -14935.052,E2 -14935.052} C_VEL
LIN {X 0,Y 325.662,Z 586.761,A -85,B 0,C 180,E1 -14936.288,E2 -14936.288} C_VEL
LIN {X 0,Y 325.271,Z 586.859,A -85,B 0,C 180,E1 -14938.762,E2 -14938.762} C_VEL
LIN {X 0,Y 325.185,Z 586.317,A -85,B 0,C 180,E1 -14940,E2 -14940} C_VEL
LIN {X 0,Y 325.141,Z 585.346,A -85,B 0,C 180,E1 -14941.239,E2 -14941.239} C_VEL
LIN {X 0,Y 325.14,Z 583.944,A -85,B 0,C 180,E1 -14942.478,E2 -14942.478} C_VEL
LIN {X 0,Y 325.266,Z 581.048,A -85,B 0,C 180,E1 -14944.337,E2 -14944.337} C_VEL
LIN {X 0,Y 325.462,Z 577.115,A -85,B 0,C 180,E1 -14946.199,E2 -14946.199} C_VEL
LIN {X 0,Y 325.784,Z 572.042,A -85,B 0,C 180,E1 -14948.061,E2 -14948.061} C_VEL
LIN {X 0,Y 326.289,Z 565.691,A -85,B 0,C 180,E1 -14949.923,E2 -14949.923} C_VEL
LIN {X 0,Y 327.008,Z 557.829,A -85,B 0,C 180,E1 -14951.781,E2 -14951.781} C_VEL
LIN {X 0,Y 327.89,Z 548.049,A -85,B 0,C 180,E1 -14953.638,E2 -14953.638} C_VEL
LIN {X 0,Y 328.863,Z 538.112,A -85,B 0,C 180,E1 -14955.177,E2 -14955.177} C_VEL
LIN {X 0,Y 329.705,Z 527.589,A -85,B 0,C 180,E1 -14956.508,E2 -14956.508} C_VEL
LIN {X 0,Y 330.687,Z 515.021,A -85,B 0,C 180,E1 -14957.789,E2 -14957.789} C_VEL
LIN {X 0,Y 330.93,Z 509.621,A -85,B 0,C 180,E1 -14958.255,E2 -14958.255} C_VEL
LIN {X 0,Y 328.172,Z 496.109,A -85,B 0,C 180,E1 -14959.33,E2 -14959.33} C_VEL
LIN {X 0,Y 325.475,Z 482.705,A -85,B 0,C 180,E1 -14960.149,E2 -14960.149} C_VEL
LIN {X 0,Y 325.351,Z 481.841,A -85,B 0,C 180,E1 -14960.22,E2 -14960.22} C_VEL
LIN {X 0,Y 325.422,Z 478.081,A -85,B 0,C 180,E1 -14964.226,E2 -14964.226} C_VEL
LIN {X 0,Y 325.593,Z 475.931,A -85,B 0,C 180,E1 -14966.955,E2 -14966.955} C_VEL
LIN {X 0,Y 325.987,Z 475.881,A -85,B 0,C 180,E1 -14970.416,E2 -14970.416} C_VEL
LIN {X 0,Y 326.33,Z 475.836,A -85,B 0,C 180,E1 -14974.053,E2 -14974.053} C_VEL
LIN {X 0,Y 326.607,Z 475.798,A -85,B 0,C 180,E1 -14977.233,E2 -14977.233} C_VEL
LIN {X 0,Y 326.595,Z 475.805,A -85,B 0,C 180,E1 -14980.209,E2 -14980.209} C_VEL
LIN {X 0,Y 326.566,Z 475.804,A -85,B 0,C 180,E1 -14983.526,E2 -14983.526} C_VEL
LIN {X 0,Y 326.58,Z 475.802,A -85,B 0,C 180,E1 -14987.028,E2 -14987.028} C_VEL
LIN {X 0,Y 326.616,Z 475.798,A -85,B 0,C 180,E1 -14990.773,E2 -14990.773} C_VEL
LIN {X 0,Y 326.617,Z 475.8,A -85,B 0,C 180,E1 -14994.481,E2 -14994.481} C_VEL
LIN {X 0,Y 326.614,Z 475.798,A -85,B 0,C 180,E1 -14997.456,E2 -14997.456} C_VEL
LIN {X 0,Y 326.652,Z 475.797,A -85,B 0,C 180,E1 -15000.34,E2 -15000.34} C_VEL
LIN {X 0,Y 326.695,Z 475.79,A -85,B 0,C 180,E1 -15004.516,E2 -15004.516} C_VEL
LIN {X 0,Y 326.651,Z 475.795,A -85,B 0,C 180,E1 -15008.545,E2 -15008.545} C_VEL
LIN {X 0,Y 326.749,Z 475.781,A -85,B 0,C 180,E1 -15011.177,E2 -15011.177} C_VEL
LIN {X 0,Y 326.768,Z 475.779,A -85,B 0,C 180,E1 -15015.433,E2 -15015.433} C_VEL
LIN {X 0,Y 326.775,Z 475.778,A -85,B 0,C 180,E1 -15018.839,E2 -15018.839} C_VEL
LIN {X 0,Y 326.961,Z 475.755,A -85,B 0,C 180,E1 -15022.59,E2 -15022.59} C_VEL
LIN {X 0,Y 326.78,Z 475.777,A -85,B 0,C 180,E1 -15025.065,E2 -15025.065} C_VEL
LIN {X 0,Y 327.051,Z 475.745,A -85,B 0,C 180,E1 -15027.537,E2 -15027.537} C_VEL
LIN {X 0,Y 327.203,Z 475.73,A -85,B 0,C 180,E1 -15030,E2 -15030} C_VEL
LIN {X 0,Y 327.05,Z 475.745,A -85,B 0,C 180,E1 -15032.463,E2 -15032.463} C_VEL
LIN {X 0,Y 326.959,Z 475.758,A -85,B 0,C 180,E1 -15036.17,E2 -15036.17} C_VEL
LIN {X 0,Y 326.81,Z 475.779,A -85,B 0,C 180,E1 -15039.906,E2 -15039.906} C_VEL
LIN {X 0,Y 326.764,Z 475.782,A -85,B 0,C 180,E1 -15043.685,E2 -15043.685} C_VEL
LIN {X 0,Y 326.704,Z 475.789,A -85,B 0,C 180,E1 -15047.527,E2 -15047.527} C_VEL
LIN {X 0,Y 326.669,Z 475.794,A -85,B 0,C 180,E1 -15050.134,E2 -15050.134} C_VEL
LIN {X 0,Y 326.656,Z 475.795,A -85,B 0,C 180,E1 -15054.128,E2 -15054.128} C_VEL
LIN {X 0,Y 326.686,Z 475.788,A -85,B 0,C 180,E1 -15056.857,E2 -15056.857} C_VEL
LIN {X 0,Y 326.637,Z 475.795,A -85,B 0,C 180,E1 -15060.609,E2 -15060.609} C_VEL
LIN {X 0,Y 326.611,Z 475.802,A -85,B 0,C 180,E1 -15064.019,E2 -15064.019} C_VEL
LIN {X 0,Y 326.632,Z 475.796,A -85,B 0,C 180,E1 -15067.239,E2 -15067.239} C_VEL
LIN {X 0,Y 326.58,Z 475.802,A -85,B 0,C 180,E1 -15071.131,E2 -15071.131} C_VEL
LIN {X 0,Y 326.53,Z 475.808,A -85,B 0,C 180,E1 -15074.742,E2 -15074.742} C_VEL
LIN {X 0,Y 326.578,Z 475.804,A -85,B 0,C 180,E1 -15078.154,E2 -15078.154} C_VEL
LIN {X 0,Y 326.625,Z 475.799,A -85,B 0,C 180,E1 -15081.391,E2 -15081.391} C_VEL
LIN {X 0,Y 326.621,Z 475.797,A -85,B 0,C 180,E1 -15084.851,E2 -15084.851} C_VEL
LIN {X 0,Y 326.611,Z 475.801,A -85,B 0,C 180,E1 -15087.455,E2 -15087.455} C_VEL
LIN {X 0,Y 326.662,Z 475.792,A -85,B 0,C 180,E1 -15090.341,E2 -15090.341} C_VEL
LIN {X 0,Y 326.691,Z 475.788,A -85,B 0,C 180,E1 -15094.516,E2 -15094.516} C_VEL
LIN {X 0,Y 326.648,Z 475.793,A -85,B 0,C 180,E1 -15098.545,E2 -15098.545} C_VEL
LIN {X 0,Y 326.736,Z 475.783,A -85,B 0,C 180,E1 -15101.279,E2 -15101.279} C_VEL
LIN {X 0,Y 326.019,Z 475.872,A -85,B 0,C 180,E1 -15102.308,E2 -15102.308} C_VEL
LIN {X 0,Y 323.179,Z 476.227,A -85,B 0,C 180,E1 -15103.984,E2 -15103.984} C_VEL
LIN {X 0,Y 320.799,Z 476.525,A -85,B 0,C 180,E1 -15105.342,E2 -15105.342} C_VEL
LIN {X 0,Y 319.773,Z 476.65,A -85,B 0,C 180,E1 -15106.392,E2 -15106.392} C_VEL
LIN {X 0,Y 319.685,Z 476.661,A -85,B 0,C 180,E1 -15106.748,E2 -15106.748} C_VEL
LIN {X 0,Y 319.759,Z 476.654,A -85,B 0,C 180,E1 -15109.873,E2 -15109.873} C_VEL
LIN {X 0,Y 319.934,Z 476.629,A -85,B 0,C 180,E1 -15112.426,E2 -15112.426} C_VEL
LIN {X 0,Y 319.748,Z 476.654,A -85,B 0,C 180,E1 -15114.956,E2 -15114.956} C_VEL
LIN {X 0,Y 319.992,Z 476.628,A -85,B 0,C 180,E1 -15117.482,E2 -15117.482} C_VEL
LIN {X 0,Y 320.151,Z 476.604,A -85,B 0,C 180,E1 -15120,E2 -15120} C_VEL
LIN {X 0,Y 319.99,Z 476.622,A -85,B 0,C 180,E1 -15122.517,E2 -15122.517} C_VEL
LIN {X 0,Y 319.952,Z 476.627,A -85,B 0,C 180,E1 -15126.305,E2 -15126.305} C_VEL
LIN {X 0,Y 319.843,Z 476.642,A -85,B 0,C 180,E1 -15128.848,E2 -15128.848} C_VEL
LIN {X 0,Y 319.682,Z 476.661,A -85,B 0,C 180,E1 -15132.7,E2 -15132.7} C_VEL
LIN {X 0,Y 319.699,Z 476.663,A -85,B 0,C 180,E1 -15135.295,E2 -15135.295} C_VEL
LIN {X 0,Y 319.674,Z 476.666,A -85,B 0,C 180,E1 -15139.255,E2 -15139.255} C_VEL
LIN {X 0,Y 319.57,Z 476.68,A -85,B 0,C 180,E1 -15143.319,E2 -15143.319} C_VEL
LIN {X 0,Y 319.618,Z 476.669,A -85,B 0,C 180,E1 -15146.089,E2 -15146.089} C_VEL
LIN {X 0,Y 319.579,Z 476.676,A -85,B 0,C 180,E1 -15148.934,E2 -15148.934} C_VEL
LIN {X 0,Y 319.531,Z 476.681,A -85,B 0,C 180,E1 -15151.862,E2 -15151.862} C_VEL
LIN {X 0,Y 319.58,Z 476.677,A -85,B 0,C 180,E1 -15155.543,E2 -15155.543} C_VEL
LIN {X 0,Y 319.583,Z 476.673,A -85,B 0,C 180,E1 -15158.007,E2 -15158.007} C_VEL
LIN {X 0,Y 319.597,Z 476.674,A -85,B 0,C 180,E1 -15161.612,E2 -15161.612} C_VEL
LIN {X 0,Y 319.648,Z 476.706,A -85,B 0,C 180,E1 -15164.373,E2 -15164.373} C_VEL
LIN {X 0,Y 320.618,Z 482.277,A -85,B 0,C 180,E1 -15168.183,E2 -15168.183} C_VEL
LIN {X 0,Y 321.599,Z 487.949,A -85,B 0,C 180,E1 -15171.88,E2 -15171.88} C_VEL
LIN {X 0,Y 321.781,Z 491.219,A -85,B 0,C 180,E1 -15173.912,E2 -15173.912} C_VEL
LIN {X 0,Y 321.181,Z 496.121,A -85,B 0,C 180,E1 -15176.836,E2 -15176.836} C_VEL
LIN {X 0,Y 320.189,Z 503.512,A -85,B 0,C 180,E1 -15181.126,E2 -15181.126} C_VEL
LIN {X 0,Y 319.31,Z 510.806,A -85,B 0,C 180,E1 -15185.28,E2 -15185.28} C_VEL
LIN {X 0,Y 318.669,Z 518.127,A -85,B 0,C 180,E1 -15189.405,E2 -15189.405} C_VEL
LIN {X 0,Y 320.085,Z 531.776,A -85,B 0,C 180,E1 -15190.154,E2 -15190.154} C_VEL
LIN {X 0,Y 321.457,Z 544.715,A -85,B 0,C 180,E1 -15191.105,E2 -15191.105} C_VEL
LIN {X 0,Y 322.627,Z 556.99,A -85,B 0,C 180,E1 -15192.244,E2 -15192.244} C_VEL
LIN {X 0,Y 322.146,Z 564.335,A -85,B 0,C 180,E1 -15193.035,E2 -15193.035} C_VEL
LIN {X 0,Y 320.974,Z 576.141,A -85,B 0,C 180,E1 -15194.557,E2 -15194.557} C_VEL
LIN {X 0,Y 320.116,Z 585.366,A -85,B 0,C 180,E1 -15196.025,E2 -15196.025} C_VEL
LIN {X 0,Y 319.266,Z 595.078,A -85,B 0,C 180,E1 -15197.929,E2 -15197.929} C_VEL
LIN {X 0,Y 318.614,Z 602.927,A -85,B 0,C 180,E1 -15199.836,E2 -15199.836} C_VEL
LIN {X 0,Y 318.261,Z 609.19,A -85,B 0,C 180,E1 -15201.748,E2 -15201.748} C_VEL
LIN {X 0,Y 318.064,Z 614.672,A -85,B 0,C 180,E1 -15203.896,E2 -15203.896} C_VEL
LIN {X 0,Y 318.045,Z 617.919,A -85,B 0,C 180,E1 -15205.565,E2 -15205.565} C_VEL
LIN {X 0,Y 318.043,Z 620.607,A -85,B 0,C 180,E1 -15207.467,E2 -15207.467} C_VEL
LIN {X 0,Y 318.173,Z 621.836,A -85,B 0,C 180,E1 -15208.735,E2 -15208.735} C_VEL
LIN {X 0,Y 318.161,Z 622.628,A -85,B 0,C 180,E1 -15210,E2 -15210} C_VEL
LIN {X 0,Y 318.091,Z 622.973,A -85,B 0,C 180,E1 -15211.266,E2 -15211.266} C_VEL
LIN {X 0,Y 317.903,Z 622.366,A -85,B 0,C 180,E1 -15213.803,E2 -15213.803} C_VEL
LIN {X 0,Y 317.859,Z 620.795,A -85,B 0,C 180,E1 -15215.749,E2 -15215.749} C_VEL
LIN {X 0,Y 318.201,Z 617.364,A -85,B 0,C 180,E1 -15218.254,E2 -15218.254} C_VEL
LIN {X 0,Y 318.72,Z 613.587,A -85,B 0,C 180,E1 -15220.161,E2 -15220.161} C_VEL
LIN {X 0,Y 319.456,Z 608.793,A -85,B 0,C 180,E1 -15222.064,E2 -15222.064} C_VEL
LIN {X 0,Y 320.974,Z 601.747,A -85,B 0,C 180,E1 -15224.261,E2 -15224.261} C_VEL
LIN {X 0,Y 322.635,Z 592.942,A -85,B 0,C 180,E1 -15226.45,E2 -15226.45} C_VEL
LIN {X 0,Y 324.859,Z 583.712,A -85,B 0,C 180,E1 -15228.282,E2 -15228.282} C_VEL
LIN {X 0,Y 327.356,Z 572.514,A -85,B 0,C 180,E1 -15230.091,E2 -15230.091} C_VEL
LIN {X 0,Y 328.786,Z 565.913,A -85,B 0,C 180,E1 -15230.98,E2 -15230.98} C_VEL
LIN {X 0,Y 329.665,Z 553.926,A -85,B 0,C 180,E1 -15232.566,E2 -15232.566} C_VEL
LIN {X 0,Y 329.001,Z 543.139,A -85,B 0,C 180,E1 -15233.946,E2 -15233.946} C_VEL
LIN {X 0,Y 327.004,Z 531.325,A -85,B 0,C 180,E1 -15235.489,E2 -15235.489} C_VEL
LIN {X 0,Y 324.304,Z 521.265,A -85,B 0,C 180,E1 -15236.883,E2 -15236.883} C_VEL
LIN {X 0,Y 322.248,Z 514.884,A -85,B 0,C 180,E1 -15237.805,E2 -15237.805} C_VEL
LIN {X 0,Y 320.86,Z 511.294,A -85,B 0,C 180,E1 -15238.375,E2 -15238.375} C_VEL
LIN {X 0,Y 320.674,Z 509.93,A -85,B 0,C 180,E1 -15238.548,E2 -15238.548} C_VEL
LIN {X 0,Y 321.562,Z 505.554,A -85,B 0,C 180,E1 -15241.638,E2 -15241.638} C_VEL
LIN {X 0,Y 322.397,Z 501.874,A -85,B 0,C 180,E1 -15244.526,E2 -15244.526} C_VEL
LIN {X 0,Y 322.885,Z 499.768,A -85,B 0,C 180,E1 -15246.356,E2 -15246.356} C_VEL
LIN {X 0,Y 323.018,Z 497.058,A -85,B 0,C 180,E1 -15249.122,E2 -15249.122} C_VEL
LIN {X 0,Y 322.706,Z 494.487,A -85,B 0,C 180,E1 -15252.465,E2 -15252.465} C_VEL
LIN {X 0,Y 322.398,Z 492.593,A -85,B 0,C 180,E1 -15255.767,E2 -15255.767} C_VEL
LIN {X 0,Y 322.094,Z 491.311,A -85,B 0,C 180,E1 -15259.111,E2 -15259.111} C_VEL
LIN {X 0,Y 321.879,Z 490.628,A -85,B 0,C 180,E1 -15262.312,E2 -15262.312} C_VEL
LIN {X 0,Y 321.498,Z 490.497,A -85,B 0,C 180,E1 -15265.364,E2 -15265.364} C_VEL
LIN {X 0,Y 321.033,Z 490.811,A -85,B 0,C 180,E1 -15268.626,E2 -15268.626} C_VEL
LIN {X 0,Y 320.611,Z 491.592,A -85,B 0,C 180,E1 -15271.659,E2 -15271.659} C_VEL
LIN {X 0,Y 321.486,Z 493.977,A -85,B 0,C 180,E1 -15272.062,E2 -15272.062} C_VEL
LIN {X 0,Y 323.187,Z 496.505,A -85,B 0,C 180,E1 -15272.673,E2 -15272.673} C_VEL
LIN {X 0,Y 328.138,Z 506.358,A -85,B 0,C 180,E1 -15274.637,E2 -15274.637} C_VEL
LIN {X 0,Y 331.567,Z 515.511,A -85,B 0,C 180,E1 -15276.251,E2 -15276.251} C_VEL
LIN {X 0,Y 333.441,Z 522.7,A -85,B 0,C 180,E1 -15277.447,E2 -15277.447} C_VEL
LIN {X 0,Y 333.906,Z 525.155,A -85,B 0,C 180,E1 -15277.836,E2 -15277.836} C_VEL
LIN {X 0,Y 331.617,Z 536.591,A -85,B 0,C 180,E1 -15279.23,E2 -15279.23} C_VEL
LIN {X 0,Y 328.993,Z 548.165,A -85,B 0,C 180,E1 -15280.988,E2 -15280.988} C_VEL
LIN {X 0,Y 326.576,Z 557.714,A -85,B 0,C 180,E1 -15282.788,E2 -15282.788} C_VEL
LIN {X 0,Y 324.619,Z 565.474,A -85,B 0,C 180,E1 -15284.621,E2 -15284.621} C_VEL
LIN {X 0,Y 322.692,Z 572.729,A -85,B 0,C 180,E1 -15286.781,E2 -15286.781} C_VEL
LIN {X 0,Y 321.255,Z 577.688,A -85,B 0,C 180,E1 -15288.645,E2 -15288.645} C_VEL
LIN {X 0,Y 320.306,Z 581.519,A -85,B 0,C 180,E1 -15290.529,E2 -15290.529} C_VEL
LIN {X 0,Y 319.347,Z 584.394,A -85,B 0,C 180,E1 -15292.413,E2 -15292.413} C_VEL
LIN {X 0,Y 318.946,Z 585.794,A -85,B 0,C 180,E1 -15293.675,E2 -15293.675} C_VEL
LIN {X 0,Y 318.851,Z 586.763,A -85,B 0,C 180,E1 -15294.942,E2 -15294.942} C_VEL
LIN {X 0,Y 318.607,Z 587.321,A -85,B 0,C 180,E1 -15296.206,E2 -15296.206} C_VEL
LIN {X 0,Y 318.198,Z 587.283,A -85,B 0,C 180,E1 -15298.735,E2 -15298.735} C_VEL
LIN {X 0,Y 318.094,Z 586.658,A -85,B 0,C 180,E1 -15300,E2 -15300} C_VEL
LIN {X 0,Y 318.046,Z 585.593,A -85,B 0,C 180,E1 -15301.267,E2 -15301.267} C_VEL
LIN {X 0,Y 318.05,Z 584.125,A -85,B 0,C 180,E1 -15302.533,E2 -15302.533} C_VEL
LIN {X 0,Y 318.204,Z 581.103,A -85,B 0,C 180,E1 -15304.434,E2 -15304.434} C_VEL
LIN {X 0,Y 318.385,Z 577.034,A -85,B 0,C 180,E1 -15306.337,E2 -15306.337} C_VEL
LIN {X 0,Y 318.718,Z 571.813,A -85,B 0,C 180,E1 -15308.241,E2 -15308.241} C_VEL
LIN {X 0,Y 319.275,Z 565.308,A -85,B 0,C 180,E1 -15310.143,E2 -15310.143} C_VEL
LIN {X 0,Y 319.998,Z 557.226,A -85,B 0,C 180,E1 -15312.043,E2 -15312.043} C_VEL
LIN {X 0,Y 320.95,Z 547.296,A -85,B 0,C 180,E1 -15313.938,E2 -15313.938} C_VEL
LIN {X 0,Y 321.993,Z 537.096,A -85,B 0,C 180,E1 -15315.509,E2 -15315.509} C_VEL
LIN {X 0,Y 322.947,Z 525.014,A -85,B 0,C 180,E1 -15317.02,E2 -15317.02} C_VEL
LIN {X 0,Y 323.838,Z 513.306,A -85,B 0,C 180,E1 -15318.178,E2 -15318.178} C_VEL
LIN {X 0,Y 323.98,Z 511.502,A -85,B 0,C 180,E1 -15318.334,E2 -15318.334} C_VEL
LIN {X 0,Y 321.737,Z 499.611,A -85,B 0,C 180,E1 -15319.348,E2 -15319.348} C_VEL
LIN {X 0,Y 318.906,Z 485.439,A -85,B 0,C 180,E1 -15320.274,E2 -15320.274} C_VEL
LIN {X 0,Y 318.281,Z 482.214,A -85,B 0,C 180,E1 -15320.48,E2 -15320.48} C_VEL
LIN {X 0,Y 318.393,Z 478.212,A -85,B 0,C 180,E1 -15324.797,E2 -15324.797} C_VEL
LIN {X 0,Y 318.446,Z 476.95,A -85,B 0,C 180,E1 -15326.193,E2 -15326.193} C_VEL
LIN {X 0,Y 318.775,Z 476.774,A -85,B 0,C 180,E1 -15329.015,E2 -15329.015} C_VEL
LIN {X 0,Y 319.086,Z 476.737,A -85,B 0,C 180,E1 -15331.912,E2 -15331.912} C_VEL
LIN {X 0,Y 319.437,Z 476.692,A -85,B 0,C 180,E1 -15335.506,E2 -15335.506} C_VEL
LIN {X 0,Y 319.533,Z 476.682,A -85,B 0,C 180,E1 -15338.014,E2 -15338.014} C_VEL
LIN {X 0,Y 319.53,Z 476.68,A -85,B 0,C 180,E1 -15341.597,E2 -15341.597} C_VEL
LIN {X 0,Y 319.492,Z 476.684,A -85,B 0,C 180,E1 -15345.257,E2 -15345.257} C_VEL
LIN {X 0,Y 319.533,Z 476.681,A -85,B 0,C 180,E1 -15348.712,E2 -15348.712} C_VEL
LIN {X 0,Y 319.582,Z 476.678,A -85,B 0,C 180,E1 -15352.344,E2 -15352.344} C_VEL
LIN {X 0,Y 319.565,Z 476.675,A -85,B 0,C 180,E1 -15355.124,E2 -15355.124} C_VEL
LIN {X 0,Y 319.571,Z 476.675,A -85,B 0,C 180,E1 -15359.059,E2 -15359.059} C_VEL
LIN {X 0,Y 319.61,Z 476.672,A -85,B 0,C 180,E1 -15362.498,E2 -15362.498} C_VEL
LIN {X 0,Y 319.61,Z 476.67,A -85,B 0,C 180,E1 -15365.304,E2 -15365.304} C_VEL
LIN {X 0,Y 319.602,Z 476.676,A -85,B 0,C 180,E1 -15368.048,E2 -15368.048} C_VEL
LIN {X 0,Y 319.694,Z 476.659,A -85,B 0,C 180,E1 -15370.962,E2 -15370.962} C_VEL
LIN {X 0,Y 319.736,Z 476.654,A -85,B 0,C 180,E1 -15375.276,E2 -15375.276} C_VEL
LIN {X 0,Y 319.757,Z 476.655,A -85,B 0,C 180,E1 -15379.873,E2 -15379.873} C_VEL
LIN {X 0,Y 319.916,Z 476.634,A -85,B 0,C 180,E1 -15382.426,E2 -15382.426} C_VEL
LIN {X 0,Y 319.749,Z 476.652,A -85,B 0,C 180,E1 -15384.956,E2 -15384.956} C_VEL
LIN {X 0,Y 319.995,Z 476.623,A -85,B 0,C 180,E1 -15387.482,E2 -15387.482} C_VEL
LIN {X 0,Y 320.154,Z 476.608,A -85,B 0,C 180,E1 -15390,E2 -15390} C_VEL
LIN {X 0,Y 319.994,Z 476.623,A -85,B 0,C 180,E1 -15392.517,E2 -15392.517} C_VEL
LIN {X 0,Y 319.916,Z 476.634,A -85,B 0,C 180,E1 -15396.306,E2 -15396.306} C_VEL
LIN {X 0,Y 319.757,Z 476.655,A -85,B 0,C 180,E1 -15400.127,E2 -15400.127} C_VEL
LIN {X 0,Y 319.735,Z 476.654,A -85,B 0,C 180,E1 -15404.724,E2 -15404.724} C_VEL
LIN {X 0,Y 319.693,Z 476.659,A -85,B 0,C 180,E1 -15409.038,E2 -15409.038} C_VEL
LIN {X 0,Y 319.574,Z 476.675,A -85,B 0,C 180,E1 -15413.319,E2 -15413.319} C_VEL
LIN {X 0,Y 319.637,Z 476.67,A -85,B 0,C 180,E1 -15416.088,E2 -15416.088} C_VEL
LIN {X 0,Y 319.583,Z 476.673,A -85,B 0,C 180,E1 -15418.934,E2 -15418.934} C_VEL
LIN {X 0,Y 319.535,Z 476.685,A -85,B 0,C 180,E1 -15421.861,E2 -15421.861} C_VEL
LIN {X 0,Y 319.583,Z 476.676,A -85,B 0,C 180,E1 -15425.543,E2 -15425.543} C_VEL
LIN {X 0,Y 319.577,Z 476.677,A -85,B 0,C 180,E1 -15428.007,E2 -15428.007} C_VEL
LIN {X 0,Y 319.528,Z 476.684,A -85,B 0,C 180,E1 -15431.597,E2 -15431.597} C_VEL
LIN {X 0,Y 319.491,Z 476.686,A -85,B 0,C 180,E1 -15435.257,E2 -15435.257} C_VEL
LIN {X 0,Y 319.53,Z 476.68,A -85,B 0,C 180,E1 -15438.711,E2 -15438.711} C_VEL
LIN {X 0,Y 319.563,Z 476.676,A -85,B 0,C 180,E1 -15442.347,E2 -15442.347} C_VEL
LIN {X 0,Y 319.562,Z 476.677,A -85,B 0,C 180,E1 -15445.123,E2 -15445.123} C_VEL
LIN {X 0,Y 319.571,Z 476.675,A -85,B 0,C 180,E1 -15449.057,E2 -15449.057} C_VEL
LIN {X 0,Y 319.61,Z 476.67,A -85,B 0,C 180,E1 -15452.498,E2 -15452.498} C_VEL
LIN {X 0,Y 319.606,Z 476.673,A -85,B 0,C 180,E1 -15455.304,E2 -15455.304} C_VEL
LIN {X 0,Y 319.598,Z 476.673,A -85,B 0,C 180,E1 -15458.047,E2 -15458.047} C_VEL
LIN {X 0,Y 319.67,Z 476.662,A -85,B 0,C 180,E1 -15461.267,E2 -15461.267} C_VEL
LIN {X 0,Y 319.732,Z 476.657,A -85,B 0,C 180,E1 -15465.275,E2 -15465.275} C_VEL
LIN {X 0,Y 319.685,Z 476.661,A -85,B 0,C 180,E1 -15466.748,E2 -15466.748} C_VEL
LIN {X 0,Y 319.03,Z 476.746,A -85,B 0,C 180,E1 -15467.799,E2 -15467.799} C_VEL
LIN {X 0,Y 316.283,Z 477.09,A -85,B 0,C 180,E1 -15469.513,E2 -15469.513} C_VEL
LIN {X 0,Y 313.959,Z 477.377,A -85,B 0,C 180,E1 -15470.902,E2 -15470.902} C_VEL
LIN {X 0,Y 312.956,Z 477.501,A -85,B 0,C 180,E1 -15471.975,E2 -15471.975} C_VEL
LIN {X 0,Y 312.87,Z 477.509,A -85,B 0,C 180,E1 -15472.338,E2 -15472.338} C_VEL
LIN {X 0,Y 312.718,Z 477.529,A -85,B 0,C 180,E1 -15474.842,E2 -15474.842} C_VEL
LIN {X 0,Y 312.992,Z 477.495,A -85,B 0,C 180,E1 -15478.713,E2 -15478.713} C_VEL
LIN {X 0,Y 312.991,Z 477.498,A -85,B 0,C 180,E1 -15481.286,E2 -15481.286} C_VEL
LIN {X 0,Y 312.718,Z 477.531,A -85,B 0,C 180,E1 -15485.157,E2 -15485.157} C_VEL
LIN {X 0,Y 312.872,Z 477.512,A -85,B 0,C 180,E1 -15487.745,E2 -15487.745} C_VEL
LIN {X 0,Y 312.669,Z 477.538,A -85,B 0,C 180,E1 -15491.671,E2 -15491.671} C_VEL
LIN {X 0,Y 312.7,Z 477.532,A -85,B 0,C 180,E1 -15494.888,E2 -15494.888} C_VEL
LIN {X 0,Y 312.63,Z 477.543,A -85,B 0,C 180,E1 -15499.236,E2 -15499.236} C_VEL
LIN {X 0,Y 312.546,Z 477.551,A -85,B 0,C 180,E1 -15502.789,E2 -15502.789} C_VEL
LIN {X 0,Y 312.596,Z 477.544,A -85,B 0,C 180,E1 -15505.933,E2 -15505.933} C_VEL
LIN {X 0,Y 312.538,Z 477.553,A -85,B 0,C 180,E1 -15509.651,E2 -15509.651} C_VEL
LIN {X 0,Y 312.519,Z 477.555,A -85,B 0,C 180,E1 -15513.689,E2 -15513.689} C_VEL
LIN {X 0,Y 312.541,Z 477.555,A -85,B 0,C 180,E1 -15517.383,E2 -15517.383} C_VEL
LIN {X 0,Y 312.526,Z 477.553,A -85,B 0,C 180,E1 -15520.703,E2 -15520.703} C_VEL
LIN {X 0,Y 312.598,Z 477.567,A -85,B 0,C 180,E1 -15524.183,E2 -15524.183} C_VEL
LIN {X 0,Y 313.465,Z 482.625,A -85,B 0,C 180,E1 -15527.731,E2 -15527.731} C_VEL
LIN {X 0,Y 314.441,Z 488.209,A -85,B 0,C 180,E1 -15531.47,E2 -15531.47} C_VEL
LIN {X 0,Y 314.758,Z 491.357,A -85,B 0,C 180,E1 -15533.496,E2 -15533.496} C_VEL
LIN {X 0,Y 314.328,Z 495.466,A -85,B 0,C 180,E1 -15536.016,E2 -15536.016} C_VEL
LIN {X 0,Y 313.269,Z 502.838,A -85,B 0,C 180,E1 -15540.426,E2 -15540.426} C_VEL
LIN {X 0,Y 312.324,Z 510.102,A -85,B 0,C 180,E1 -15544.689,E2 -15544.689} C_VEL
LIN {X 0,Y 311.61,Z 517.727,A -85,B 0,C 180,E1 -15549.107,E2 -15549.107} C_VEL
LIN {X 0,Y 312.098,Z 523.593,A -85,B 0,C 180,E1 -15549.443,E2 -15549.443} C_VEL
LIN {X 0,Y 313.617,Z 537.782,A -85,B 0,C 180,E1 -15550.358,E2 -15550.358} C_VEL
LIN {X 0,Y 315.011,Z 550.712,A -85,B 0,C 180,E1 -15551.463,E2 -15551.463} C_VEL
LIN {X 0,Y 315.629,Z 559.257,A -85,B 0,C 180,E1 -15552.339,E2 -15552.339} C_VEL
LIN {X 0,Y 314.386,Z 571.635,A -85,B 0,C 180,E1 -15553.841,E2 -15553.841} C_VEL
LIN {X 0,Y 313.381,Z 581.802,A -85,B 0,C 180,E1 -15555.387,E2 -15555.387} C_VEL
LIN {X 0,Y 312.416,Z 592.159,A -85,B 0,C 180,E1 -15557.33,E2 -15557.33} C_VEL
LIN {X 0,Y 311.663,Z 600.426,A -85,B 0,C 180,E1 -15559.279,E2 -15559.279} C_VEL
LIN {X 0,Y 311.264,Z 607.117,A -85,B 0,C 180,E1 -15561.234,E2 -15561.234} C_VEL
LIN {X 0,Y 311.018,Z 613.209,A -85,B 0,C 180,E1 -15563.513,E2 -15563.513} C_VEL
LIN {X 0,Y 310.99,Z 617.104,A -85,B 0,C 180,E1 -15565.464,E2 -15565.464} C_VEL
LIN {X 0,Y 310.96,Z 619.901,A -85,B 0,C 180,E1 -15567.41,E2 -15567.41} C_VEL
LIN {X 0,Y 311.114,Z 621.187,A -85,B 0,C 180,E1 -15568.706,E2 -15568.706} C_VEL
LIN {X 0,Y 311.104,Z 622.035,A -85,B 0,C 180,E1 -15570,E2 -15570} C_VEL
LIN {X 0,Y 311.013,Z 622.46,A -85,B 0,C 180,E1 -15571.295,E2 -15571.295} C_VEL
LIN {X 0,Y 310.817,Z 622.44,A -85,B 0,C 180,E1 -15572.592,E2 -15572.592} C_VEL
LIN {X 0,Y 310.828,Z 621.999,A -85,B 0,C 180,E1 -15573.89,E2 -15573.89} C_VEL
LIN {X 0,Y 310.828,Z 619.909,A -85,B 0,C 180,E1 -15576.492,E2 -15576.492} C_VEL
LIN {X 0,Y 311.145,Z 617.237,A -85,B 0,C 180,E1 -15578.443,E2 -15578.443} C_VEL
LIN {X 0,Y 311.693,Z 613.624,A -85,B 0,C 180,E1 -15580.392,E2 -15580.392} C_VEL
LIN {X 0,Y 312.508,Z 608.985,A -85,B 0,C 180,E1 -15582.336,E2 -15582.336} C_VEL
LIN {X 0,Y 314.117,Z 602.174,A -85,B 0,C 180,E1 -15584.579,E2 -15584.579} C_VEL
LIN {X 0,Y 315.683,Z 594.622,A -85,B 0,C 180,E1 -15586.589,E2 -15586.589} C_VEL
LIN {X 0,Y 318.2,Z 584.743,A -85,B 0,C 180,E1 -15588.679,E2 -15588.679} C_VEL
LIN {X 0,Y 320.823,Z 573.976,A -85,B 0,C 180,E1 -15590.518,E2 -15590.518} C_VEL
LIN {X 0,Y 322.507,Z 566.687,A -85,B 0,C 180,E1 -15591.576,E2 -15591.576} C_VEL
LIN {X 0,Y 323.465,Z 556.209,A -85,B 0,C 180,E1 -15593.023,E2 -15593.023} C_VEL
LIN {X 0,Y 323.154,Z 546.181,A -85,B 0,C 180,E1 -15594.407,E2 -15594.407} C_VEL
LIN {X 0,Y 321.337,Z 533.855,A -85,B 0,C 180,E1 -15596.133,E2 -15596.133} C_VEL
LIN {X 0,Y 318.985,Z 524.261,A -85,B 0,C 180,E1 -15597.561,E2 -15597.561} C_VEL
LIN {X 0,Y 315.801,Z 514.263,A -85,B 0,C 180,E1 -15599.18,E2 -15599.18} C_VEL
LIN {X 0,Y 314.301,Z 510.492,A -85,B 0,C 180,E1 -15599.876,E2 -15599.876} C_VEL
LIN {X 0,Y 314.079,Z 508.92,A -85,B 0,C 180,E1 -15600.128,E2 -15600.128} C_VEL
LIN {X 0,Y 314.767,Z 505.895,A -85,B 0,C 180,E1 -15602.403,E2 -15602.403} C_VEL
LIN {X 0,Y 315.641,Z 502.317,A -85,B 0,C 180,E1 -15605.374,E2 -15605.374} C_VEL
LIN {X 0,Y 315.97,Z 500.66,A -85,B 0,C 180,E1 -15606.91,E2 -15606.91} C_VEL
LIN {X 0,Y 316.111,Z 498.758,A -85,B 0,C 180,E1 -15608.909,E2 -15608.909} C_VEL
LIN {X 0,Y 315.819,Z 496.457,A -85,B 0,C 180,E1 -15611.882,E2 -15611.882} C_VEL
LIN {X 0,Y 315.493,Z 494.334,A -85,B 0,C 180,E1 -15615.467,E2 -15615.467} C_VEL
LIN {X 0,Y 315.169,Z 492.842,A -85,B 0,C 180,E1 -15619.304,E2 -15619.304} C_VEL
LIN {X 0,Y 314.859,Z 492.135,A -85,B 0,C 180,E1 -15622.939,E2 -15622.939} C_VEL
LIN {X 0,Y 314.522,Z 492.039,A -85,B 0,C 180,E1 -15626.039,E2 -15626.039} C_VEL
LIN {X 0,Y 313.859,Z 492.559,A -85,B 0,C 180,E1 -15630.053,E2 -15630.053} C_VEL
LIN {X 0,Y 314.841,Z 495.215,A -85,B 0,C 180,E1 -15630.588,E2 -15630.588} C_VEL
LIN {X 0,Y 316.557,Z 497.166,A -85,B 0,C 180,E1 -15631.235,E2 -15631.235} C_VEL
LIN {X 0,Y 317.121,Z 498.733,A -85,B 0,C 180,E1 -15631.544,E2 -15631.544} C_VEL
LIN {X 0,Y 321.771,Z 507.645,A -85,B 0,C 180,E1 -15633.574,E2 -15633.574} C_VEL
LIN {X 0,Y 325.083,Z 516.081,A -85,B 0,C 180,E1 -15635.232,E2 -15635.232} C_VEL
LIN {X 0,Y 327.406,Z 524.34,A -85,B 0,C 180,E1 -15636.731,E2 -15636.731} C_VEL
LIN {X 0,Y 327.961,Z 527.716,A -85,B 0,C 180,E1 -15637.311,E2 -15637.311} C_VEL
LIN {X 0,Y 325.09,Z 540.306,A -85,B 0,C 180,E1 -15638.936,E2 -15638.936} C_VEL
LIN {X 0,Y 322.556,Z 550.474,A -85,B 0,C 180,E1 -15640.593,E2 -15640.593} C_VEL
LIN {X 0,Y 320.028,Z 559.597,A -85,B 0,C 180,E1 -15642.425,E2 -15642.425} C_VEL
LIN {X 0,Y 317.621,Z 568.199,A -85,B 0,C 180,E1 -15644.602,E2 -15644.602} C_VEL
LIN {X 0,Y 315.923,Z 574.094,A -85,B 0,C 180,E1 -15646.492,E2 -15646.492} C_VEL
LIN {X 0,Y 314.418,Z 578.839,A -85,B 0,C 180,E1 -15648.395,E2 -15648.395} C_VEL
LIN {X 0,Y 313.378,Z 582.528,A -85,B 0,C 180,E1 -15650.317,E2 -15650.317} C_VEL
LIN {X 0,Y 312.379,Z 585.25,A -85,B 0,C 180,E1 -15652.242,E2 -15652.242} C_VEL
LIN {X 0,Y 311.924,Z 586.549,A -85,B 0,C 180,E1 -15653.532,E2 -15653.532} C_VEL
LIN {X 0,Y 311.805,Z 587.389,A -85,B 0,C 180,E1 -15654.828,E2 -15654.828} C_VEL
LIN {X 0,Y 311.555,Z 587.878,A -85,B 0,C 180,E1 -15656.12,E2 -15656.12} C_VEL
LIN {X 0,Y 311.295,Z 587.987,A -85,B 0,C 180,E1 -15657.412,E2 -15657.412} C_VEL
LIN {X 0,Y 311.112,Z 587.688,A -85,B 0,C 180,E1 -15658.706,E2 -15658.706} C_VEL
LIN {X 0,Y 311,Z 586.95,A -85,B 0,C 180,E1 -15660,E2 -15660} C_VEL
LIN {X 0,Y 310.95,Z 585.818,A -85,B 0,C 180,E1 -15661.295,E2 -15661.295} C_VEL
LIN {X 0,Y 310.963,Z 584.285,A -85,B 0,C 180,E1 -15662.591,E2 -15662.591} C_VEL
LIN {X 0,Y 311.123,Z 581.144,A -85,B 0,C 180,E1 -15664.535,E2 -15664.535} C_VEL
LIN {X 0,Y 311.365,Z 576.385,A -85,B 0,C 180,E1 -15666.707,E2 -15666.707} C_VEL
LIN {X 0,Y 311.762,Z 570.529,A -85,B 0,C 180,E1 -15668.753,E2 -15668.753} C_VEL
LIN {X 0,Y 312.343,Z 563.582,A -85,B 0,C 180,E1 -15670.698,E2 -15670.698} C_VEL
LIN {X 0,Y 313.129,Z 555.042,A -85,B 0,C 180,E1 -15672.641,E2 -15672.641} C_VEL
LIN {X 0,Y 314.215,Z 544.423,A -85,B 0,C 180,E1 -15674.574,E2 -15674.574} C_VEL
LIN {X 0,Y 315.25,Z 534.07,A -85,B 0,C 180,E1 -15676.107,E2 -15676.107} C_VEL
LIN {X 0,Y 316.132,Z 522.778,A -85,B 0,C 180,E1 -15677.465,E2 -15677.465} C_VEL
LIN {X 0,Y 316.881,Z 513.069,A -85,B 0,C 180,E1 -15678.424,E2 -15678.424} C_VEL
LIN {X 0,Y 315.993,Z 506.975,A -85,B 0,C 180,E1 -15678.983,E2 -15678.983} C_VEL
LIN {X 0,Y 313.62,Z 494.814,A -85,B 0,C 180,E1 -15679.948,E2 -15679.948} C_VEL
LIN {X 0,Y 311.208,Z 482.619,A -85,B 0,C 180,E1 -15680.705,E2 -15680.705} C_VEL
LIN {X 0,Y 311.244,Z 479.61,A -85,B 0,C 180,E1 -15683.982,E2 -15683.982} C_VEL
LIN {X 0,Y 311.361,Z 478.273,A -85,B 0,C 180,E1 -15685.46,E2 -15685.46} C_VEL
LIN {X 0,Y 311.476,Z 477.689,A -85,B 0,C 180,E1 -15686.826,E2 -15686.826} C_VEL
LIN {X 0,Y 311.798,Z 477.644,A -85,B 0,C 180,E1 -15689.729,E2 -15689.729} C_VEL
LIN {X 0,Y 312.09,Z 477.608,A -85,B 0,C 180,E1 -15692.716,E2 -15692.716} C_VEL
LIN {X 0,Y 312.429,Z 477.567,A -85,B 0,C 180,E1 -15695.922,E2 -15695.922} C_VEL
LIN {X 0,Y 312.48,Z 477.558,A -85,B 0,C 180,E1 -15699.032,E2 -15699.032} C_VEL
LIN {X 0,Y 312.494,Z 477.56,A -85,B 0,C 180,E1 -15702.432,E2 -15702.432} C_VEL
LIN {X 0,Y 312.462,Z 477.564,A -85,B 0,C 180,E1 -15706.035,E2 -15706.035} C_VEL
LIN {X 0,Y 312.508,Z 477.557,A -85,B 0,C 180,E1 -15709.875,E2 -15709.875} C_VEL
LIN {X 0,Y 312.542,Z 477.552,A -85,B 0,C 180,E1 -15712.617,E2 -15712.617} C_VEL
LIN {X 0,Y 312.524,Z 477.557,A -85,B 0,C 180,E1 -15716.311,E2 -15716.311} C_VEL
LIN {X 0,Y 312.543,Z 477.554,A -85,B 0,C 180,E1 -15720.349,E2 -15720.349} C_VEL
LIN {X 0,Y 312.607,Z 477.547,A -85,B 0,C 180,E1 -15724.064,E2 -15724.064} C_VEL
LIN {X 0,Y 312.592,Z 477.545,A -85,B 0,C 180,E1 -15727.529,E2 -15727.529} C_VEL
LIN {X 0,Y 312.644,Z 477.539,A -85,B 0,C 180,E1 -15731.656,E2 -15731.656} C_VEL
LIN {X 0,Y 312.699,Z 477.533,A -85,B 0,C 180,E1 -15735.686,E2 -15735.686} C_VEL
LIN {X 0,Y 312.703,Z 477.532,A -85,B 0,C 180,E1 -15739.642,E2 -15739.642} C_VEL
LIN {X 0,Y 312.857,Z 477.515,A -85,B 0,C 180,E1 -15742.254,E2 -15742.254} C_VEL
LIN {X 0,Y 312.719,Z 477.528,A -85,B 0,C 180,E1 -15744.842,E2 -15744.842} C_VEL
LIN {X 0,Y 312.994,Z 477.494,A -85,B 0,C 180,E1 -15748.713,E2 -15748.713} C_VEL
LIN {X 0,Y 312.996,Z 477.494,A -85,B 0,C 180,E1 -15751.286,E2 -15751.286} C_VEL
LIN {X 0,Y 312.712,Z 477.529,A -85,B 0,C 180,E1 -15755.157,E2 -15755.157} C_VEL
LIN {X 0,Y 312.823,Z 477.519,A -85,B 0,C 180,E1 -15757.747,E2 -15757.747} C_VEL
LIN {X 0,Y 312.674,Z 477.537,A -85,B 0,C 180,E1 -15761.671,E2 -15761.671} C_VEL
LIN {X 0,Y 312.704,Z 477.53,A -85,B 0,C 180,E1 -15764.887,E2 -15764.887} C_VEL
LIN {X 0,Y 312.635,Z 477.539,A -85,B 0,C 180,E1 -15769.236,E2 -15769.236} C_VEL
LIN {X 0,Y 312.55,Z 477.549,A -85,B 0,C 180,E1 -15772.789,E2 -15772.789} C_VEL
LIN {X 0,Y 312.606,Z 477.547,A -85,B 0,C 180,E1 -15775.935,E2 -15775.935} C_VEL
LIN {X 0,Y 312.541,Z 477.554,A -85,B 0,C 180,E1 -15779.65,E2 -15779.65} C_VEL
LIN {X 0,Y 312.522,Z 477.557,A -85,B 0,C 180,E1 -15783.688,E2 -15783.688} C_VEL
LIN {X 0,Y 312.541,Z 477.552,A -85,B 0,C 180,E1 -15787.383,E2 -15787.383} C_VEL
LIN {X 0,Y 312.492,Z 477.556,A -85,B 0,C 180,E1 -15790.709,E2 -15790.709} C_VEL
LIN {X 0,Y 312.454,Z 477.563,A -85,B 0,C 180,E1 -15794.209,E2 -15794.209} C_VEL
LIN {X 0,Y 312.486,Z 477.561,A -85,B 0,C 180,E1 -15797.918,E2 -15797.918} C_VEL
LIN {X 0,Y 312.536,Z 477.555,A -85,B 0,C 180,E1 -15801.91,E2 -15801.91} C_VEL
LIN {X 0,Y 312.508,Z 477.559,A -85,B 0,C 180,E1 -15805.79,E2 -15805.79} C_VEL
LIN {X 0,Y 312.525,Z 477.552,A -85,B 0,C 180,E1 -15808.854,E2 -15808.854} C_VEL
LIN {X 0,Y 312.575,Z 477.55,A -85,B 0,C 180,E1 -15811.824,E2 -15811.824} C_VEL
LIN {X 0,Y 312.587,Z 477.544,A -85,B 0,C 180,E1 -15814.711,E2 -15814.711} C_VEL
LIN {X 0,Y 312.588,Z 477.549,A -85,B 0,C 180,E1 -15817.529,E2 -15817.529} C_VEL
LIN {X 0,Y 312.639,Z 477.543,A -85,B 0,C 180,E1 -15821.656,E2 -15821.656} C_VEL
LIN {X 0,Y 312.694,Z 477.536,A -85,B 0,C 180,E1 -15825.686,E2 -15825.686} C_VEL
LIN {X 0,Y 312.703,Z 477.535,A -85,B 0,C 180,E1 -15829.642,E2 -15829.642} C_VEL
LIN {X 0,Y 312.87,Z 477.509,A -85,B 0,C 180,E1 -15832.338,E2 -15832.338} C_VEL
LIN {X 0,Y 312.19,Z 477.598,A -85,B 0,C 180,E1 -15833.411,E2 -15833.411} C_VEL
LIN {X 0,Y 309.338,Z 477.951,A -85,B 0,C 180,E1 -15835.158,E2 -15835.158} C_VEL
LIN {X 0,Y 306.953,Z 478.249,A -85,B 0,C 180,E1 -15836.574,E2 -15836.574} C_VEL
LIN {X 0,Y 305.965,Z 478.374,A -85,B 0,C 180,E1 -15837.671,E2 -15837.671} C_VEL
LIN {X 0,Y 305.903,Z 478.377,A -85,B 0,C 180,E1 -15838.042,E2 -15838.042} C_VEL
LIN {X 0,Y 306.056,Z 478.359,A -85,B 0,C 180,E1 -15840,E2 -15840} C_VEL
LIN {X 0,Y 305.886,Z 478.379,A -85,B 0,C 180,E1 -15842.633,E2 -15842.633} C_VEL
LIN {X 0,Y 305.853,Z 478.384,A -85,B 0,C 180,E1 -15846.597,E2 -15846.597} C_VEL
LIN {X 0,Y 305.736,Z 478.402,A -85,B 0,C 180,E1 -15849.259,E2 -15849.259} C_VEL
LIN {X 0,Y 305.589,Z 478.42,A -85,B 0,C 180,E1 -15853.296,E2 -15853.296} C_VEL
LIN {X 0,Y 305.594,Z 478.417,A -85,B 0,C 180,E1 -15856.02,E2 -15856.02} C_VEL
LIN {X 0,Y 305.577,Z 478.423,A -85,B 0,C 180,E1 -15859.445,E2 -15859.445} C_VEL
LIN {X 0,Y 305.49,Z 478.431,A -85,B 0,C 180,E1 -15863.041,E2 -15863.041} C_VEL
LIN {X 0,Y 305.525,Z 478.424,A -85,B 0,C 180,E1 -15866.219,E2 -15866.219} C_VEL
LIN {X 0,Y 305.488,Z 478.431,A -85,B 0,C 180,E1 -15869.047,E2 -15869.047} C_VEL
LIN {X 0,Y 305.442,Z 478.436,A -85,B 0,C 180,E1 -15871.952,E2 -15871.952} C_VEL
LIN {X 0,Y 305.463,Z 478.436,A -85,B 0,C 180,E1 -15875.113,E2 -15875.113} C_VEL
LIN {X 0,Y 305.483,Z 478.43,A -85,B 0,C 180,E1 -15878.537,E2 -15878.537} C_VEL
LIN {X 0,Y 305.514,Z 478.426,A -85,B 0,C 180,E1 -15882.598,E2 -15882.598} C_VEL
LIN {X 0,Y 305.549,Z 478.558,A -85,B 0,C 180,E1 -15884.097,E2 -15884.097} C_VEL
LIN {X 0,Y 306.612,Z 484.484,A -85,B 0,C 180,E1 -15888.339,E2 -15888.339} C_VEL
LIN {X 0,Y 307.515,Z 489.718,A -85,B 0,C 180,E1 -15891.898,E2 -15891.898} C_VEL
LIN {X 0,Y 307.687,Z 492.277,A -85,B 0,C 180,E1 -15893.568,E2 -15893.568} C_VEL
LIN {X 0,Y 307.065,Z 497.239,A -85,B 0,C 180,E1 -15896.681,E2 -15896.681} C_VEL
LIN {X 0,Y 305.995,Z 504.57,A -85,B 0,C 180,E1 -15901.163,E2 -15901.163} C_VEL
LIN {X 0,Y 305.065,Z 511.771,A -85,B 0,C 180,E1 -15905.501,E2 -15905.501} C_VEL
LIN {X 0,Y 304.536,Z 517.42,A -85,B 0,C 180,E1 -15908.864,E2 -15908.864} C_VEL
LIN {X 0,Y 305.99,Z 532.384,A -85,B 0,C 180,E1 -15909.76,E2 -15909.76} C_VEL
LIN {X 0,Y 307.453,Z 546.53,A -85,B 0,C 180,E1 -15910.898,E2 -15910.898} C_VEL
LIN {X 0,Y 308.509,Z 558.232,A -85,B 0,C 180,E1 -15912.089,E2 -15912.089} C_VEL
LIN {X 0,Y 307.578,Z 569.044,A -85,B 0,C 180,E1 -15913.405,E2 -15913.405} C_VEL
LIN {X 0,Y 306.413,Z 580.184,A -85,B 0,C 180,E1 -15915.073,E2 -15915.073} C_VEL
LIN {X 0,Y 305.443,Z 590.589,A -85,B 0,C 180,E1 -15917.036,E2 -15917.036} C_VEL
LIN {X 0,Y 304.653,Z 599.104,A -85,B 0,C 180,E1 -15919.029,E2 -15919.029} C_VEL
LIN {X 0,Y 304.238,Z 605.941,A -85,B 0,C 180,E1 -15921.03,E2 -15921.03} C_VEL
LIN {X 0,Y 303.97,Z 612.197,A -85,B 0,C 180,E1 -15923.362,E2 -15923.362} C_VEL
LIN {X 0,Y 303.936,Z 616.231,A -85,B 0,C 180,E1 -15925.358,E2 -15925.358} C_VEL
LIN {X 0,Y 303.884,Z 619.13,A -85,B 0,C 180,E1 -15927.349,E2 -15927.349} C_VEL
LIN {X 0,Y 304.055,Z 620.517,A -85,B 0,C 180,E1 -15928.676,E2 -15928.676} C_VEL
LIN {X 0,Y 304.049,Z 621.423,A -85,B 0,C 180,E1 -15930,E2 -15930} C_VEL
LIN {X 0,Y 303.937,Z 621.908,A -85,B 0,C 180,E1 -15931.325,E2 -15931.325} C_VEL
LIN {X 0,Y 303.735,Z 621.979,A -85,B 0,C 180,E1 -15932.653,E2 -15932.653} C_VEL
LIN {X 0,Y 303.732,Z 621.632,A -85,B 0,C 180,E1 -15933.981,E2 -15933.981} C_VEL
LIN {X 0,Y 303.742,Z 619.672,A -85,B 0,C 180,E1 -15936.644,E2 -15936.644} C_VEL
LIN {X 0,Y 303.951,Z 618.107,A -85,B 0,C 180,E1 -15937.975,E2 -15937.975} C_VEL
LIN {X 0,Y 304.446,Z 614.946,A -85,B 0,C 180,E1 -15939.97,E2 -15939.97} C_VEL
LIN {X 0,Y 305.208,Z 610.795,A -85,B 0,C 180,E1 -15941.961,E2 -15941.961} C_VEL
LIN {X 0,Y 306.484,Z 605.643,A -85,B 0,C 180,E1 -15943.933,E2 -15943.933} C_VEL
LIN {X 0,Y 308.26,Z 598.18,A -85,B 0,C 180,E1 -15946.218,E2 -15946.218} C_VEL
LIN {X 0,Y 310.434,Z 589.914,A -85,B 0,C 180,E1 -15948.231,E2 -15948.231} C_VEL
LIN {X 0,Y 312.923,Z 580.908,A -85,B 0,C 180,E1 -15950.03,E2 -15950.03} C_VEL
LIN {X 0,Y 315.371,Z 571.561,A -85,B 0,C 180,E1 -15951.574,E2 -15951.574} C_VEL
LIN {X 0,Y 316.419,Z 566.402,A -85,B 0,C 180,E1 -15952.357,E2 -15952.357} C_VEL
LIN {X 0,Y 317.375,Z 557.347,A -85,B 0,C 180,E1 -15953.686,E2 -15953.686} C_VEL
LIN {X 0,Y 317.1,Z 546.318,A -85,B 0,C 180,E1 -15955.301,E2 -15955.301} C_VEL
LIN {X 0,Y 315.264,Z 534.023,A -85,B 0,C 180,E1 -15957.172,E2 -15957.172} C_VEL
LIN {X 0,Y 312.845,Z 524,A -85,B 0,C 180,E1 -15958.821,E2 -15958.821} C_VEL
LIN {X 0,Y 309.509,Z 513.564,A -85,B 0,C 180,E1 -15960.74,E2 -15960.74} C_VEL
LIN {X 0,Y 308.061,Z 510.32,A -85,B 0,C 180,E1 -15961.48,E2 -15961.48} C_VEL
LIN {X 0,Y 307.623,Z 507.933,A -85,B 0,C 180,E1 -15961.863,E2 -15961.863} C_VEL
LIN {X 0,Y 308.548,Z 504.271,A -85,B 0,C 180,E1 -15964.916,E2 -15964.916} C_VEL
LIN {X 0,Y 309.08,Z 501.227,A -85,B 0,C 180,E1 -15967.875,E2 -15967.875} C_VEL
LIN {X 0,Y 309.131,Z 499.769,A -85,B 0,C 180,E1 -15969.537,E2 -15969.537} C_VEL
LIN {X 0,Y 308.8,Z 497.142,A -85,B 0,C 180,E1 -15973.257,E2 -15973.257} C_VEL
LIN {X 0,Y 308.461,Z 495.303,A -85,B 0,C 180,E1 -15976.881,E2 -15976.881} C_VEL
LIN {X 0,Y 308.105,Z 494.062,A -85,B 0,C 180,E1 -15980.856,E2 -15980.856} C_VEL
LIN {X 0,Y 307.879,Z 493.65,A -85,B 0,C 180,E1 -15983.594,E2 -15983.594} C_VEL
LIN {X 0,Y 307.441,Z 493.625,A -85,B 0,C 180,E1 -15986.727,E2 -15986.727} C_VEL
LIN {X 0,Y 307.223,Z 493.827,A -85,B 0,C 180,E1 -15988.22,E2 -15988.22} C_VEL
LIN {X 0,Y 308.296,Z 496.499,A -85,B 0,C 180,E1 -15988.879,E2 -15988.879} C_VEL
LIN {X 0,Y 309.8,Z 498.213,A -85,B 0,C 180,E1 -15989.549,E2 -15989.549} C_VEL
LIN {X 0,Y 310.903,Z 500.676,A -85,B 0,C 180,E1 -15990.178,E2 -15990.178} C_VEL
LIN {X 0,Y 312.358,Z 502.462,A -85,B 0,C 180,E1 -15990.782,E2 -15990.782} C_VEL
LIN {X 0,Y 317.563,Z 513.758,A -85,B 0,C 180,E1 -15993.462,E2 -15993.462} C_VEL
LIN {X 0,Y 320.65,Z 523.14,A -85,B 0,C 180,E1 -15995.39,E2 -15995.39} C_VEL
LIN {X 0,Y 321.885,Z 528.892,A -85,B 0,C 180,E1 -15996.496,E2 -15996.496} C_VEL
LIN {X 0,Y 322.039,Z 530.319,A -85,B 0,C 180,E1 -15996.747,E2 -15996.747} C_VEL
LIN {X 0,Y 319.614,Z 540.114,A -85,B 0,C 180,E1 -15998.049,E2 -15998.049} C_VEL
LIN {X 0,Y 316.629,Z 551.122,A -85,B 0,C 180,E1 -15999.877,E2 -15999.877} C_VEL
LIN {X 0,Y 313.946,Z 560.24,A -85,B 0,C 180,E1 -16001.736,E2 -16001.736} C_VEL
LIN {X 0,Y 311.674,Z 567.616,A -85,B 0,C 180,E1 -16003.629,E2 -16003.629} C_VEL
LIN {X 0,Y 309.713,Z 573.695,A -85,B 0,C 180,E1 -16005.546,E2 -16005.546} C_VEL
LIN {X 0,Y 308.166,Z 578.596,A -85,B 0,C 180,E1 -16007.488,E2 -16007.488} C_VEL
LIN {X 0,Y 306.837,Z 582.438,A -85,B 0,C 180,E1 -16009.442,E2 -16009.442} C_VEL
LIN {X 0,Y 306.058,Z 584.672,A -85,B 0,C 180,E1 -16010.9,E2 -16010.9} C_VEL
LIN {X 0,Y 305.395,Z 586.099,A -85,B 0,C 180,E1 -16012.064,E2 -16012.064} C_VEL
LIN {X 0,Y 304.903,Z 587.275,A -85,B 0,C 180,E1 -16013.382,E2 -16013.382} C_VEL
LIN {X 0,Y 304.746,Z 588.043,A -85,B 0,C 180,E1 -16014.707,E2 -16014.707} C_VEL
LIN {X 0,Y 304.505,Z 588.447,A -85,B 0,C 180,E1 -16016.03,E2 -16016.03} C_VEL
LIN {X 0,Y 304.218,Z 588.464,A -85,B 0,C 180,E1 -16017.352,E2 -16017.352} C_VEL
LIN {X 0,Y 304.023,Z 588.047,A -85,B 0,C 180,E1 -16018.676,E2 -16018.676} C_VEL
LIN {X 0,Y 303.906,Z 587.237,A -85,B 0,C 180,E1 -16020,E2 -16020} C_VEL
LIN {X 0,Y 303.854,Z 586.033,A -85,B 0,C 180,E1 -16021.326,E2 -16021.326} C_VEL
LIN {X 0,Y 303.916,Z 583.405,A -85,B 0,C 180,E1 -16023.315,E2 -16023.315} C_VEL
LIN {X 0,Y 304.1,Z 579.777,A -85,B 0,C 180,E1 -16025.305,E2 -16025.305} C_VEL
LIN {X 0,Y 304.424,Z 574.819,A -85,B 0,C 180,E1 -16027.381,E2 -16027.381} C_VEL
LIN {X 0,Y 304.899,Z 567.971,A -85,B 0,C 180,E1 -16029.62,E2 -16029.62} C_VEL
LIN {X 0,Y 305.596,Z 560.359,A -85,B 0,C 180,E1 -16031.609,E2 -16031.609} C_VEL
LIN {X 0,Y 306.521,Z 550.939,A -85,B 0,C 180,E1 -16033.593,E2 -16033.593} C_VEL
LIN {X 0,Y 307.554,Z 540.274,A -85,B 0,C 180,E1 -16035.406,E2 -16035.406} C_VEL
LIN {X 0,Y 308.457,Z 530.879,A -85,B 0,C 180,E1 -16036.72,E2 -16036.72} C_VEL
LIN {X 0,Y 309.435,Z 519.519,A -85,B 0,C 180,E1 -16038.027,E2 -16038.027} C_VEL
LIN {X 0,Y 309.847,Z 513.018,A -85,B 0,C 180,E1 -16038.659,E2 -16038.659} C_VEL
LIN {X 0,Y 307.772,Z 501.825,A -85,B 0,C 180,E1 -16039.674,E2 -16039.674} C_VEL
LIN {X 0,Y 305.116,Z 488.134,A -85,B 0,C 180,E1 -16040.658,E2 -16040.658} C_VEL
LIN {X 0,Y 304.143,Z 482.976,A -85,B 0,C 180,E1 -16040.988,E2 -16040.988} C_VEL
LIN {X 0,Y 304.316,Z 478.681,A -85,B 0,C 180,E1 -16045.751,E2 -16045.751} C_VEL
LIN {X 0,Y 304.663,Z 478.533,A -85,B 0,C 180,E1 -16048.976,E2 -16048.976} C_VEL
LIN {X 0,Y 304.97,Z 478.496,A -85,B 0,C 180,E1 -16052.008,E2 -16052.008} C_VEL
LIN {X 0,Y 305.276,Z 478.456,A -85,B 0,C 180,E1 -16055.138,E2 -16055.138} C_VEL
LIN {X 0,Y 305.428,Z 478.44,A -85,B 0,C 180,E1 -16058.523,E2 -16058.523} C_VEL
LIN {X 0,Y 305.444,Z 478.436,A -85,B 0,C 180,E1 -16061.857,E2 -16061.857} C_VEL
LIN {X 0,Y 305.404,Z 478.44,A -85,B 0,C 180,E1 -16065.511,E2 -16065.511} C_VEL
LIN {X 0,Y 305.445,Z 478.439,A -85,B 0,C 180,E1 -16068.143,E2 -16068.143} C_VEL
LIN {X 0,Y 305.499,Z 478.428,A -85,B 0,C 180,E1 -16071.601,E2 -16071.601} C_VEL
LIN {X 0,Y 305.467,Z 478.432,A -85,B 0,C 180,E1 -16074.887,E2 -16074.887} C_VEL
LIN {X 0,Y 305.455,Z 478.436,A -85,B 0,C 180,E1 -16078.355,E2 -16078.355} C_VEL
LIN {X 0,Y 305.517,Z 478.425,A -85,B 0,C 180,E1 -16081.113,E2 -16081.113} C_VEL
LIN {X 0,Y 305.576,Z 478.423,A -85,B 0,C 180,E1 -16084.088,E2 -16084.088} C_VEL
LIN {X 0,Y 305.505,Z 478.429,A -85,B 0,C 180,E1 -16088.403,E2 -16088.403} C_VEL
LIN {X 0,Y 305.595,Z 478.416,A -85,B 0,C 180,E1 -16091.218,E2 -16091.218} C_VEL
LIN {X 0,Y 305.654,Z 478.409,A -85,B 0,C 180,E1 -16095.349,E2 -16095.349} C_VEL
LIN {X 0,Y 305.64,Z 478.411,A -85,B 0,C 180,E1 -16099.399,E2 -16099.399} C_VEL
LIN {X 0,Y 305.801,Z 478.395,A -85,B 0,C 180,E1 -16102.074,E2 -16102.074} C_VEL
LIN {X 0,Y 305.69,Z 478.404,A -85,B 0,C 180,E1 -16104.723,E2 -16104.723} C_VEL
LIN {X 0,Y 305.961,Z 478.371,A -85,B 0,C 180,E1 -16108.683,E2 -16108.683} C_VEL
LIN {X 0,Y 305.962,Z 478.371,A -85,B 0,C 180,E1 -16111.316,E2 -16111.316} C_VEL
LIN {X 0,Y 305.68,Z 478.405,A -85,B 0,C 180,E1 -16115.276,E2 -16115.276} C_VEL
LIN {X 0,Y 305.77,Z 478.399,A -85,B 0,C 180,E1 -16117.927,E2 -16117.927} C_VEL
LIN {X 0,Y 305.608,Z 478.419,A -85,B 0,C 180,E1 -16121.945,E2 -16121.945} C_VEL
LIN {X 0,Y 305.642,Z 478.41,A -85,B 0,C 180,E1 -16125.035,E2 -16125.035} C_VEL
LIN {X 0,Y 305.581,Z 478.419,A -85,B 0,C 180,E1 -16129.445,E2 -16129.445} C_VEL
LIN {X 0,Y 305.494,Z 478.428,A -85,B 0,C 180,E1 -16133.041,E2 -16133.041} C_VEL
LIN {X 0,Y 305.535,Z 478.426,A -85,B 0,C 180,E1 -16136.221,E2 -16136.221} C_VEL
LIN {X 0,Y 305.491,Z 478.429,A -85,B 0,C 180,E1 -16139.047,E2 -16139.047} C_VEL
LIN {X 0,Y 305.446,Z 478.438,A -85,B 0,C 180,E1 -16141.952,E2 -16141.952} C_VEL
LIN {X 0,Y 305.466,Z 478.432,A -85,B 0,C 180,E1 -16145.112,E2 -16145.112} C_VEL
LIN {X 0,Y 305.47,Z 478.431,A -85,B 0,C 180,E1 -16148.533,E2 -16148.533} C_VEL
LIN {X 0,Y 305.457,Z 478.433,A -85,B 0,C 180,E1 -16152.585,E2 -16152.585} C_VEL
LIN {X 0,Y 305.428,Z 478.437,A -85,B 0,C 180,E1 -16156.345,E2 -16156.345} C_VEL
LIN {X 0,Y 305.46,Z 478.436,A -85,B 0,C 180,E1 -16159.892,E2 -16159.892} C_VEL
LIN {X 0,Y 305.483,Z 478.435,A -85,B 0,C 180,E1 -16163.631,E2 -16163.631} C_VEL
LIN {X 0,Y 305.466,Z 478.431,A -85,B 0,C 180,E1 -16166.483,E2 -16166.483} C_VEL
LIN {X 0,Y 305.465,Z 478.436,A -85,B 0,C 180,E1 -16169.591,E2 -16169.591} C_VEL
LIN {X 0,Y 305.522,Z 478.425,A -85,B 0,C 180,E1 -16172.608,E2 -16172.608} C_VEL
LIN {X 0,Y 305.509,Z 478.431,A -85,B 0,C 180,E1 -16175.538,E2 -16175.538} C_VEL
LIN {X 0,Y 305.521,Z 478.429,A -85,B 0,C 180,E1 -16179.815,E2 -16179.815} C_VEL
LIN {X 0,Y 305.575,Z 478.418,A -85,B 0,C 180,E1 -16182.603,E2 -16182.603} C_VEL
LIN {X 0,Y 305.65,Z 478.412,A -85,B 0,C 180,E1 -16185.349,E2 -16185.349} C_VEL
LIN {X 0,Y 305.639,Z 478.414,A -85,B 0,C 180,E1 -16189.399,E2 -16189.399} C_VEL
LIN {X 0,Y 305.808,Z 478.389,A -85,B 0,C 180,E1 -16192.336,E2 -16192.336} C_VEL
LIN {X 0,Y 305.69,Z 478.404,A -85,B 0,C 180,E1 -16194.723,E2 -16194.723} C_VEL
LIN {X 0,Y 305.903,Z 478.377,A -85,B 0,C 180,E1 -16198.042,E2 -16198.042} C_VEL
LIN {X 0,Y 305.282,Z 478.459,A -85,B 0,C 180,E1 -16199.142,E2 -16199.142} C_VEL
LIN {X 0,Y 302.411,Z 478.813,A -85,B 0,C 180,E1 -16200.93,E2 -16200.93} C_VEL
LIN {X 0,Y 299.896,Z 479.125,A -85,B 0,C 180,E1 -16202.38,E2 -16202.38} C_VEL
LIN {X 0,Y 298.747,Z 479.274,A -85,B 0,C 180,E1 -16203.504,E2 -16203.504} C_VEL
LIN {X 0,Y 298.618,Z 479.284,A -85,B 0,C 180,E1 -16203.886,E2 -16203.886} C_VEL
LIN {X 0,Y 298.798,Z 479.263,A -85,B 0,C 180,E1 -16206.754,E2 -16206.754} C_VEL
LIN {X 0,Y 298.681,Z 479.282,A -85,B 0,C 180,E1 -16209.48,E2 -16209.48} C_VEL
LIN {X 0,Y 298.552,Z 479.297,A -85,B 0,C 180,E1 -16213.615,E2 -16213.615} C_VEL
LIN {X 0,Y 298.549,Z 479.293,A -85,B 0,C 180,E1 -16216.408,E2 -16216.408} C_VEL
LIN {X 0,Y 298.511,Z 479.3,A -85,B 0,C 180,E1 -16219.655,E2 -16219.655} C_VEL
LIN {X 0,Y 298.457,Z 479.308,A -85,B 0,C 180,E1 -16223.597,E2 -16223.597} C_VEL
LIN {X 0,Y 298.485,Z 479.302,A -85,B 0,C 180,E1 -16226.575,E2 -16226.575} C_VEL
LIN {X 0,Y 298.416,Z 479.312,A -85,B 0,C 180,E1 -16229.641,E2 -16229.641} C_VEL
LIN {X 0,Y 298.395,Z 479.314,A -85,B 0,C 180,E1 -16232.8,E2 -16232.8} C_VEL
